   // GBK_TO_UNICODE[29568] := 16#D667;
   // GBK_TO_UNICODE[29569] := 16#8B0C;
   // GBK_TO_UNICODE[29570] := 16#D668;
   // GBK_TO_UNICODE[29571] := 16#8B0D;
   // GBK_TO_UNICODE[29572] := 16#D669;
   // GBK_TO_UNICODE[29573] := 16#8B0E;
   // GBK_TO_UNICODE[29574] := 16#D66A;
   // GBK_TO_UNICODE[29575] := 16#8B0F;
   // GBK_TO_UNICODE[29576] := 16#D66B;
   // GBK_TO_UNICODE[29577] := 16#8B10;
   // GBK_TO_UNICODE[29578] := 16#D66C;
   // GBK_TO_UNICODE[29579] := 16#8B11;
   // GBK_TO_UNICODE[29580] := 16#D66D;
   // GBK_TO_UNICODE[29581] := 16#8B12;
   // GBK_TO_UNICODE[29582] := 16#D66E;
   // GBK_TO_UNICODE[29583] := 16#8B13;
   // GBK_TO_UNICODE[29584] := 16#D66F;
   // GBK_TO_UNICODE[29585] := 16#8B14;
   // GBK_TO_UNICODE[29586] := 16#D670;
   // GBK_TO_UNICODE[29587] := 16#8B15;
   // GBK_TO_UNICODE[29588] := 16#D671;
   // GBK_TO_UNICODE[29589] := 16#8B16;
   // GBK_TO_UNICODE[29590] := 16#D672;
   // GBK_TO_UNICODE[29591] := 16#8B17;
   // GBK_TO_UNICODE[29592] := 16#D673;
   // GBK_TO_UNICODE[29593] := 16#8B18;
   // GBK_TO_UNICODE[29594] := 16#D674;
   // GBK_TO_UNICODE[29595] := 16#8B19;
   // GBK_TO_UNICODE[29596] := 16#D675;
   // GBK_TO_UNICODE[29597] := 16#8B1A;
   // GBK_TO_UNICODE[29598] := 16#D676;
   // GBK_TO_UNICODE[29599] := 16#8B1B;
   // GBK_TO_UNICODE[29600] := 16#D677;
   // GBK_TO_UNICODE[29601] := 16#8B1C;
   // GBK_TO_UNICODE[29602] := 16#D678;
   // GBK_TO_UNICODE[29603] := 16#8B1D;
   // GBK_TO_UNICODE[29604] := 16#D679;
   // GBK_TO_UNICODE[29605] := 16#8B1E;
   // GBK_TO_UNICODE[29606] := 16#D67A;
   // GBK_TO_UNICODE[29607] := 16#8B1F;
   // GBK_TO_UNICODE[29608] := 16#D67B;
   // GBK_TO_UNICODE[29609] := 16#8B20;
   // GBK_TO_UNICODE[29610] := 16#D67C;
   // GBK_TO_UNICODE[29611] := 16#8B21;
   // GBK_TO_UNICODE[29612] := 16#D67D;
   // GBK_TO_UNICODE[29613] := 16#8B22;
   // GBK_TO_UNICODE[29614] := 16#D67E;
   // GBK_TO_UNICODE[29615] := 16#8B23;
   // GBK_TO_UNICODE[29616] := 16#D680;
   // GBK_TO_UNICODE[29617] := 16#8B24;
   // GBK_TO_UNICODE[29618] := 16#D681;
   // GBK_TO_UNICODE[29619] := 16#8B25;
   // GBK_TO_UNICODE[29620] := 16#D682;
   // GBK_TO_UNICODE[29621] := 16#8B27;
   // GBK_TO_UNICODE[29622] := 16#D683;
   // GBK_TO_UNICODE[29623] := 16#8B28;
   // GBK_TO_UNICODE[29624] := 16#D684;
   // GBK_TO_UNICODE[29625] := 16#8B29;
   // GBK_TO_UNICODE[29626] := 16#D685;
   // GBK_TO_UNICODE[29627] := 16#8B2A;
   // GBK_TO_UNICODE[29628] := 16#D686;
   // GBK_TO_UNICODE[29629] := 16#8B2B;
   // GBK_TO_UNICODE[29630] := 16#D687;
   // GBK_TO_UNICODE[29631] := 16#8B2C;
   // GBK_TO_UNICODE[29632] := 16#D688;
   // GBK_TO_UNICODE[29633] := 16#8B2D;
   // GBK_TO_UNICODE[29634] := 16#D689;
   // GBK_TO_UNICODE[29635] := 16#8B2E;
   // GBK_TO_UNICODE[29636] := 16#D68A;
   // GBK_TO_UNICODE[29637] := 16#8B2F;
   // GBK_TO_UNICODE[29638] := 16#D68B;
   // GBK_TO_UNICODE[29639] := 16#8B30;
   // GBK_TO_UNICODE[29640] := 16#D68C;
   // GBK_TO_UNICODE[29641] := 16#8B31;
   // GBK_TO_UNICODE[29642] := 16#D68D;
   // GBK_TO_UNICODE[29643] := 16#8B32;
   // GBK_TO_UNICODE[29644] := 16#D68E;
   // GBK_TO_UNICODE[29645] := 16#8B33;
   // GBK_TO_UNICODE[29646] := 16#D68F;
   // GBK_TO_UNICODE[29647] := 16#8B34;
   // GBK_TO_UNICODE[29648] := 16#D690;
   // GBK_TO_UNICODE[29649] := 16#8B35;
   // GBK_TO_UNICODE[29650] := 16#D691;
   // GBK_TO_UNICODE[29651] := 16#8B36;
   // GBK_TO_UNICODE[29652] := 16#D692;
   // GBK_TO_UNICODE[29653] := 16#8B37;
   // GBK_TO_UNICODE[29654] := 16#D693;
   // GBK_TO_UNICODE[29655] := 16#8B38;
   // GBK_TO_UNICODE[29656] := 16#D694;
   // GBK_TO_UNICODE[29657] := 16#8B39;
   // GBK_TO_UNICODE[29658] := 16#D695;
   // GBK_TO_UNICODE[29659] := 16#8B3A;
   // GBK_TO_UNICODE[29660] := 16#D696;
   // GBK_TO_UNICODE[29661] := 16#8B3B;
   // GBK_TO_UNICODE[29662] := 16#D697;
   // GBK_TO_UNICODE[29663] := 16#8B3C;
   // GBK_TO_UNICODE[29664] := 16#D698;
   // GBK_TO_UNICODE[29665] := 16#8B3D;
   // GBK_TO_UNICODE[29666] := 16#D699;
   // GBK_TO_UNICODE[29667] := 16#8B3E;
   // GBK_TO_UNICODE[29668] := 16#D69A;
   // GBK_TO_UNICODE[29669] := 16#8B3F;
   // GBK_TO_UNICODE[29670] := 16#D69B;
   // GBK_TO_UNICODE[29671] := 16#8B40;
   // GBK_TO_UNICODE[29672] := 16#D69C;
   // GBK_TO_UNICODE[29673] := 16#8B41;
   // GBK_TO_UNICODE[29674] := 16#D69D;
   // GBK_TO_UNICODE[29675] := 16#8B42;
   // GBK_TO_UNICODE[29676] := 16#D69E;
   // GBK_TO_UNICODE[29677] := 16#8B43;
   // GBK_TO_UNICODE[29678] := 16#D69F;
   // GBK_TO_UNICODE[29679] := 16#8B44;
   // GBK_TO_UNICODE[29680] := 16#D6A0;
   // GBK_TO_UNICODE[29681] := 16#8B45;
   // GBK_TO_UNICODE[29682] := 16#D6A1;
   // GBK_TO_UNICODE[29683] := 16#5E27;
   // GBK_TO_UNICODE[29684] := 16#D6A2;
   // GBK_TO_UNICODE[29685] := 16#75C7;
   // GBK_TO_UNICODE[29686] := 16#D6A3;
   // GBK_TO_UNICODE[29687] := 16#90D1;
   // GBK_TO_UNICODE[29688] := 16#D6A4;
   // GBK_TO_UNICODE[29689] := 16#8BC1;
   // GBK_TO_UNICODE[29690] := 16#D6A5;
   // GBK_TO_UNICODE[29691] := 16#829D;
   // GBK_TO_UNICODE[29692] := 16#D6A6;
   // GBK_TO_UNICODE[29693] := 16#679D;
   // GBK_TO_UNICODE[29694] := 16#D6A7;
   // GBK_TO_UNICODE[29695] := 16#652F;
   // GBK_TO_UNICODE[29696] := 16#D6A8;
   // GBK_TO_UNICODE[29697] := 16#5431;
   // GBK_TO_UNICODE[29698] := 16#D6A9;
   // GBK_TO_UNICODE[29699] := 16#8718;
   // GBK_TO_UNICODE[29700] := 16#D6AA;
   // GBK_TO_UNICODE[29701] := 16#77E5;
   // GBK_TO_UNICODE[29702] := 16#D6AB;
   // GBK_TO_UNICODE[29703] := 16#80A2;
   // GBK_TO_UNICODE[29704] := 16#D6AC;
   // GBK_TO_UNICODE[29705] := 16#8102;
   // GBK_TO_UNICODE[29706] := 16#D6AD;
   // GBK_TO_UNICODE[29707] := 16#6C41;
   // GBK_TO_UNICODE[29708] := 16#D6AE;
   // GBK_TO_UNICODE[29709] := 16#4E4B;
   // GBK_TO_UNICODE[29710] := 16#D6AF;
   // GBK_TO_UNICODE[29711] := 16#7EC7;
   // GBK_TO_UNICODE[29712] := 16#D6B0;
   // GBK_TO_UNICODE[29713] := 16#804C;
   // GBK_TO_UNICODE[29714] := 16#D6B1;
   // GBK_TO_UNICODE[29715] := 16#76F4;
   // GBK_TO_UNICODE[29716] := 16#D6B2;
   // GBK_TO_UNICODE[29717] := 16#690D;
   // GBK_TO_UNICODE[29718] := 16#D6B3;
   // GBK_TO_UNICODE[29719] := 16#6B96;
   // GBK_TO_UNICODE[29720] := 16#D6B4;
   // GBK_TO_UNICODE[29721] := 16#6267;
   // GBK_TO_UNICODE[29722] := 16#D6B5;
   // GBK_TO_UNICODE[29723] := 16#503C;
   // GBK_TO_UNICODE[29724] := 16#D6B6;
   // GBK_TO_UNICODE[29725] := 16#4F84;
   // GBK_TO_UNICODE[29726] := 16#D6B7;
   // GBK_TO_UNICODE[29727] := 16#5740;
   // GBK_TO_UNICODE[29728] := 16#D6B8;
   // GBK_TO_UNICODE[29729] := 16#6307;
   // GBK_TO_UNICODE[29730] := 16#D6B9;
   // GBK_TO_UNICODE[29731] := 16#6B62;
   // GBK_TO_UNICODE[29732] := 16#D6BA;
   // GBK_TO_UNICODE[29733] := 16#8DBE;
   // GBK_TO_UNICODE[29734] := 16#D6BB;
   // GBK_TO_UNICODE[29735] := 16#53EA;
   // GBK_TO_UNICODE[29736] := 16#D6BC;
   // GBK_TO_UNICODE[29737] := 16#65E8;
   // GBK_TO_UNICODE[29738] := 16#D6BD;
   // GBK_TO_UNICODE[29739] := 16#7EB8;
   // GBK_TO_UNICODE[29740] := 16#D6BE;
   // GBK_TO_UNICODE[29741] := 16#5FD7;
   // GBK_TO_UNICODE[29742] := 16#D6BF;
   // GBK_TO_UNICODE[29743] := 16#631A;
   // GBK_TO_UNICODE[29744] := 16#D6C0;
   // GBK_TO_UNICODE[29745] := 16#63B7;
   // GBK_TO_UNICODE[29746] := 16#D6C1;
   // GBK_TO_UNICODE[29747] := 16#81F3;
   // GBK_TO_UNICODE[29748] := 16#D6C2;
   // GBK_TO_UNICODE[29749] := 16#81F4;
   // GBK_TO_UNICODE[29750] := 16#D6C3;
   // GBK_TO_UNICODE[29751] := 16#7F6E;
   // GBK_TO_UNICODE[29752] := 16#D6C4;
   // GBK_TO_UNICODE[29753] := 16#5E1C;
   // GBK_TO_UNICODE[29754] := 16#D6C5;
   // GBK_TO_UNICODE[29755] := 16#5CD9;
   // GBK_TO_UNICODE[29756] := 16#D6C6;
   // GBK_TO_UNICODE[29757] := 16#5236;
   // GBK_TO_UNICODE[29758] := 16#D6C7;
   // GBK_TO_UNICODE[29759] := 16#667A;
   // GBK_TO_UNICODE[29760] := 16#D6C8;
   // GBK_TO_UNICODE[29761] := 16#79E9;
   // GBK_TO_UNICODE[29762] := 16#D6C9;
   // GBK_TO_UNICODE[29763] := 16#7A1A;
   // GBK_TO_UNICODE[29764] := 16#D6CA;
   // GBK_TO_UNICODE[29765] := 16#8D28;
   // GBK_TO_UNICODE[29766] := 16#D6CB;
   // GBK_TO_UNICODE[29767] := 16#7099;
   // GBK_TO_UNICODE[29768] := 16#D6CC;
   // GBK_TO_UNICODE[29769] := 16#75D4;
   // GBK_TO_UNICODE[29770] := 16#D6CD;
   // GBK_TO_UNICODE[29771] := 16#6EDE;
   // GBK_TO_UNICODE[29772] := 16#D6CE;
   // GBK_TO_UNICODE[29773] := 16#6CBB;
   // GBK_TO_UNICODE[29774] := 16#D6CF;
   // GBK_TO_UNICODE[29775] := 16#7A92;
   // GBK_TO_UNICODE[29776] := 16#D6D0;
   // GBK_TO_UNICODE[29777] := 16#4E2D;
   // GBK_TO_UNICODE[29778] := 16#D6D1;
   // GBK_TO_UNICODE[29779] := 16#76C5;
   // GBK_TO_UNICODE[29780] := 16#D6D2;
   // GBK_TO_UNICODE[29781] := 16#5FE0;
   // GBK_TO_UNICODE[29782] := 16#D6D3;
   // GBK_TO_UNICODE[29783] := 16#949F;
   // GBK_TO_UNICODE[29784] := 16#D6D4;
   // GBK_TO_UNICODE[29785] := 16#8877;
   // GBK_TO_UNICODE[29786] := 16#D6D5;
   // GBK_TO_UNICODE[29787] := 16#7EC8;
   // GBK_TO_UNICODE[29788] := 16#D6D6;
   // GBK_TO_UNICODE[29789] := 16#79CD;
   // GBK_TO_UNICODE[29790] := 16#D6D7;
   // GBK_TO_UNICODE[29791] := 16#80BF;
   // GBK_TO_UNICODE[29792] := 16#D6D8;
   // GBK_TO_UNICODE[29793] := 16#91CD;
   // GBK_TO_UNICODE[29794] := 16#D6D9;
   // GBK_TO_UNICODE[29795] := 16#4EF2;
   // GBK_TO_UNICODE[29796] := 16#D6DA;
   // GBK_TO_UNICODE[29797] := 16#4F17;
   // GBK_TO_UNICODE[29798] := 16#D6DB;
   // GBK_TO_UNICODE[29799] := 16#821F;
   // GBK_TO_UNICODE[29800] := 16#D6DC;
   // GBK_TO_UNICODE[29801] := 16#5468;
   // GBK_TO_UNICODE[29802] := 16#D6DD;
   // GBK_TO_UNICODE[29803] := 16#5DDE;
   // GBK_TO_UNICODE[29804] := 16#D6DE;
   // GBK_TO_UNICODE[29805] := 16#6D32;
   // GBK_TO_UNICODE[29806] := 16#D6DF;
   // GBK_TO_UNICODE[29807] := 16#8BCC;
   // GBK_TO_UNICODE[29808] := 16#D6E0;
   // GBK_TO_UNICODE[29809] := 16#7CA5;
   // GBK_TO_UNICODE[29810] := 16#D6E1;
   // GBK_TO_UNICODE[29811] := 16#8F74;
   // GBK_TO_UNICODE[29812] := 16#D6E2;
   // GBK_TO_UNICODE[29813] := 16#8098;
   // GBK_TO_UNICODE[29814] := 16#D6E3;
   // GBK_TO_UNICODE[29815] := 16#5E1A;
   // GBK_TO_UNICODE[29816] := 16#D6E4;
   // GBK_TO_UNICODE[29817] := 16#5492;
   // GBK_TO_UNICODE[29818] := 16#D6E5;
   // GBK_TO_UNICODE[29819] := 16#76B1;
   // GBK_TO_UNICODE[29820] := 16#D6E6;
   // GBK_TO_UNICODE[29821] := 16#5B99;
   // GBK_TO_UNICODE[29822] := 16#D6E7;
   // GBK_TO_UNICODE[29823] := 16#663C;
   // GBK_TO_UNICODE[29824] := 16#D6E8;
   // GBK_TO_UNICODE[29825] := 16#9AA4;
   // GBK_TO_UNICODE[29826] := 16#D6E9;
   // GBK_TO_UNICODE[29827] := 16#73E0;
   // GBK_TO_UNICODE[29828] := 16#D6EA;
   // GBK_TO_UNICODE[29829] := 16#682A;
   // GBK_TO_UNICODE[29830] := 16#D6EB;
   // GBK_TO_UNICODE[29831] := 16#86DB;
   // GBK_TO_UNICODE[29832] := 16#D6EC;
   // GBK_TO_UNICODE[29833] := 16#6731;
   // GBK_TO_UNICODE[29834] := 16#D6ED;
   // GBK_TO_UNICODE[29835] := 16#732A;
   // GBK_TO_UNICODE[29836] := 16#D6EE;
   // GBK_TO_UNICODE[29837] := 16#8BF8;
   // GBK_TO_UNICODE[29838] := 16#D6EF;
   // GBK_TO_UNICODE[29839] := 16#8BDB;
   // GBK_TO_UNICODE[29840] := 16#D6F0;
   // GBK_TO_UNICODE[29841] := 16#9010;
   // GBK_TO_UNICODE[29842] := 16#D6F1;
   // GBK_TO_UNICODE[29843] := 16#7AF9;
   // GBK_TO_UNICODE[29844] := 16#D6F2;
   // GBK_TO_UNICODE[29845] := 16#70DB;
   // GBK_TO_UNICODE[29846] := 16#D6F3;
   // GBK_TO_UNICODE[29847] := 16#716E;
   // GBK_TO_UNICODE[29848] := 16#D6F4;
   // GBK_TO_UNICODE[29849] := 16#62C4;
   // GBK_TO_UNICODE[29850] := 16#D6F5;
   // GBK_TO_UNICODE[29851] := 16#77A9;
   // GBK_TO_UNICODE[29852] := 16#D6F6;
   // GBK_TO_UNICODE[29853] := 16#5631;
   // GBK_TO_UNICODE[29854] := 16#D6F7;
   // GBK_TO_UNICODE[29855] := 16#4E3B;
   // GBK_TO_UNICODE[29856] := 16#D6F8;
   // GBK_TO_UNICODE[29857] := 16#8457;
   // GBK_TO_UNICODE[29858] := 16#D6F9;
   // GBK_TO_UNICODE[29859] := 16#67F1;
   // GBK_TO_UNICODE[29860] := 16#D6FA;
   // GBK_TO_UNICODE[29861] := 16#52A9;
   // GBK_TO_UNICODE[29862] := 16#D6FB;
   // GBK_TO_UNICODE[29863] := 16#86C0;
   // GBK_TO_UNICODE[29864] := 16#D6FC;
   // GBK_TO_UNICODE[29865] := 16#8D2E;
   // GBK_TO_UNICODE[29866] := 16#D6FD;
   // GBK_TO_UNICODE[29867] := 16#94F8;
   // GBK_TO_UNICODE[29868] := 16#D6FE;
   // GBK_TO_UNICODE[29869] := 16#7B51;
   // GBK_TO_UNICODE[29870] := 16#D740;
   // GBK_TO_UNICODE[29871] := 16#8B46;
   // GBK_TO_UNICODE[29872] := 16#D741;
   // GBK_TO_UNICODE[29873] := 16#8B47;
   // GBK_TO_UNICODE[29874] := 16#D742;
   // GBK_TO_UNICODE[29875] := 16#8B48;
   // GBK_TO_UNICODE[29876] := 16#D743;
   // GBK_TO_UNICODE[29877] := 16#8B49;
   // GBK_TO_UNICODE[29878] := 16#D744;
   // GBK_TO_UNICODE[29879] := 16#8B4A;
   // GBK_TO_UNICODE[29880] := 16#D745;
   // GBK_TO_UNICODE[29881] := 16#8B4B;
   // GBK_TO_UNICODE[29882] := 16#D746;
   // GBK_TO_UNICODE[29883] := 16#8B4C;
   // GBK_TO_UNICODE[29884] := 16#D747;
   // GBK_TO_UNICODE[29885] := 16#8B4D;
   // GBK_TO_UNICODE[29886] := 16#D748;
   // GBK_TO_UNICODE[29887] := 16#8B4E;
   // GBK_TO_UNICODE[29888] := 16#D749;
   // GBK_TO_UNICODE[29889] := 16#8B4F;
   // GBK_TO_UNICODE[29890] := 16#D74A;
   // GBK_TO_UNICODE[29891] := 16#8B50;
   // GBK_TO_UNICODE[29892] := 16#D74B;
   // GBK_TO_UNICODE[29893] := 16#8B51;
   // GBK_TO_UNICODE[29894] := 16#D74C;
   // GBK_TO_UNICODE[29895] := 16#8B52;
   // GBK_TO_UNICODE[29896] := 16#D74D;
   // GBK_TO_UNICODE[29897] := 16#8B53;
   // GBK_TO_UNICODE[29898] := 16#D74E;
   // GBK_TO_UNICODE[29899] := 16#8B54;
   // GBK_TO_UNICODE[29900] := 16#D74F;
   // GBK_TO_UNICODE[29901] := 16#8B55;
   // GBK_TO_UNICODE[29902] := 16#D750;
   // GBK_TO_UNICODE[29903] := 16#8B56;
   // GBK_TO_UNICODE[29904] := 16#D751;
   // GBK_TO_UNICODE[29905] := 16#8B57;
   // GBK_TO_UNICODE[29906] := 16#D752;
   // GBK_TO_UNICODE[29907] := 16#8B58;
   // GBK_TO_UNICODE[29908] := 16#D753;
   // GBK_TO_UNICODE[29909] := 16#8B59;
   // GBK_TO_UNICODE[29910] := 16#D754;
   // GBK_TO_UNICODE[29911] := 16#8B5A;
   // GBK_TO_UNICODE[29912] := 16#D755;
   // GBK_TO_UNICODE[29913] := 16#8B5B;
   // GBK_TO_UNICODE[29914] := 16#D756;
   // GBK_TO_UNICODE[29915] := 16#8B5C;
   // GBK_TO_UNICODE[29916] := 16#D757;
   // GBK_TO_UNICODE[29917] := 16#8B5D;
   // GBK_TO_UNICODE[29918] := 16#D758;
   // GBK_TO_UNICODE[29919] := 16#8B5E;
   // GBK_TO_UNICODE[29920] := 16#D759;
   // GBK_TO_UNICODE[29921] := 16#8B5F;
   // GBK_TO_UNICODE[29922] := 16#D75A;
   // GBK_TO_UNICODE[29923] := 16#8B60;
   // GBK_TO_UNICODE[29924] := 16#D75B;
   // GBK_TO_UNICODE[29925] := 16#8B61;
   // GBK_TO_UNICODE[29926] := 16#D75C;
   // GBK_TO_UNICODE[29927] := 16#8B62;
   // GBK_TO_UNICODE[29928] := 16#D75D;
   // GBK_TO_UNICODE[29929] := 16#8B63;
   // GBK_TO_UNICODE[29930] := 16#D75E;
   // GBK_TO_UNICODE[29931] := 16#8B64;
   // GBK_TO_UNICODE[29932] := 16#D75F;
   // GBK_TO_UNICODE[29933] := 16#8B65;
   // GBK_TO_UNICODE[29934] := 16#D760;
   // GBK_TO_UNICODE[29935] := 16#8B67;
   // GBK_TO_UNICODE[29936] := 16#D761;
   // GBK_TO_UNICODE[29937] := 16#8B68;
   // GBK_TO_UNICODE[29938] := 16#D762;
   // GBK_TO_UNICODE[29939] := 16#8B69;
   // GBK_TO_UNICODE[29940] := 16#D763;
   // GBK_TO_UNICODE[29941] := 16#8B6A;
   // GBK_TO_UNICODE[29942] := 16#D764;
   // GBK_TO_UNICODE[29943] := 16#8B6B;
   // GBK_TO_UNICODE[29944] := 16#D765;
   // GBK_TO_UNICODE[29945] := 16#8B6D;
   // GBK_TO_UNICODE[29946] := 16#D766;
   // GBK_TO_UNICODE[29947] := 16#8B6E;
   // GBK_TO_UNICODE[29948] := 16#D767;
   // GBK_TO_UNICODE[29949] := 16#8B6F;
   // GBK_TO_UNICODE[29950] := 16#D768;
   // GBK_TO_UNICODE[29951] := 16#8B70;
   // GBK_TO_UNICODE[29952] := 16#D769;
   // GBK_TO_UNICODE[29953] := 16#8B71;
   // GBK_TO_UNICODE[29954] := 16#D76A;
   // GBK_TO_UNICODE[29955] := 16#8B72;
   // GBK_TO_UNICODE[29956] := 16#D76B;
   // GBK_TO_UNICODE[29957] := 16#8B73;
   // GBK_TO_UNICODE[29958] := 16#D76C;
   // GBK_TO_UNICODE[29959] := 16#8B74;
   // GBK_TO_UNICODE[29960] := 16#D76D;
   // GBK_TO_UNICODE[29961] := 16#8B75;
   // GBK_TO_UNICODE[29962] := 16#D76E;
   // GBK_TO_UNICODE[29963] := 16#8B76;
   // GBK_TO_UNICODE[29964] := 16#D76F;
   // GBK_TO_UNICODE[29965] := 16#8B77;
   // GBK_TO_UNICODE[29966] := 16#D770;
   // GBK_TO_UNICODE[29967] := 16#8B78;
   // GBK_TO_UNICODE[29968] := 16#D771;
   // GBK_TO_UNICODE[29969] := 16#8B79;
   // GBK_TO_UNICODE[29970] := 16#D772;
   // GBK_TO_UNICODE[29971] := 16#8B7A;
   // GBK_TO_UNICODE[29972] := 16#D773;
   // GBK_TO_UNICODE[29973] := 16#8B7B;
   // GBK_TO_UNICODE[29974] := 16#D774;
   // GBK_TO_UNICODE[29975] := 16#8B7C;
   // GBK_TO_UNICODE[29976] := 16#D775;
   // GBK_TO_UNICODE[29977] := 16#8B7D;
   // GBK_TO_UNICODE[29978] := 16#D776;
   // GBK_TO_UNICODE[29979] := 16#8B7E;
   // GBK_TO_UNICODE[29980] := 16#D777;
   // GBK_TO_UNICODE[29981] := 16#8B7F;
   // GBK_TO_UNICODE[29982] := 16#D778;
   // GBK_TO_UNICODE[29983] := 16#8B80;
   // GBK_TO_UNICODE[29984] := 16#D779;
   // GBK_TO_UNICODE[29985] := 16#8B81;
   // GBK_TO_UNICODE[29986] := 16#D77A;
   // GBK_TO_UNICODE[29987] := 16#8B82;
   // GBK_TO_UNICODE[29988] := 16#D77B;
   // GBK_TO_UNICODE[29989] := 16#8B83;
   // GBK_TO_UNICODE[29990] := 16#D77C;
   // GBK_TO_UNICODE[29991] := 16#8B84;
   // GBK_TO_UNICODE[29992] := 16#D77D;
   // GBK_TO_UNICODE[29993] := 16#8B85;
   // GBK_TO_UNICODE[29994] := 16#D77E;
   // GBK_TO_UNICODE[29995] := 16#8B86;
   // GBK_TO_UNICODE[29996] := 16#D780;
   // GBK_TO_UNICODE[29997] := 16#8B87;
   // GBK_TO_UNICODE[29998] := 16#D781;
   // GBK_TO_UNICODE[29999] := 16#8B88;
   // GBK_TO_UNICODE[30000] := 16#D782;
   // GBK_TO_UNICODE[30001] := 16#8B89;
   // GBK_TO_UNICODE[30002] := 16#D783;
   // GBK_TO_UNICODE[30003] := 16#8B8A;
   // GBK_TO_UNICODE[30004] := 16#D784;
   // GBK_TO_UNICODE[30005] := 16#8B8B;
   // GBK_TO_UNICODE[30006] := 16#D785;
   // GBK_TO_UNICODE[30007] := 16#8B8C;
   // GBK_TO_UNICODE[30008] := 16#D786;
   // GBK_TO_UNICODE[30009] := 16#8B8D;
   // GBK_TO_UNICODE[30010] := 16#D787;
   // GBK_TO_UNICODE[30011] := 16#8B8E;
   // GBK_TO_UNICODE[30012] := 16#D788;
   // GBK_TO_UNICODE[30013] := 16#8B8F;
   // GBK_TO_UNICODE[30014] := 16#D789;
   // GBK_TO_UNICODE[30015] := 16#8B90;
   // GBK_TO_UNICODE[30016] := 16#D78A;
   // GBK_TO_UNICODE[30017] := 16#8B91;
   // GBK_TO_UNICODE[30018] := 16#D78B;
   // GBK_TO_UNICODE[30019] := 16#8B92;
   // GBK_TO_UNICODE[30020] := 16#D78C;
   // GBK_TO_UNICODE[30021] := 16#8B93;
   // GBK_TO_UNICODE[30022] := 16#D78D;
   // GBK_TO_UNICODE[30023] := 16#8B94;
   // GBK_TO_UNICODE[30024] := 16#D78E;
   // GBK_TO_UNICODE[30025] := 16#8B95;
   // GBK_TO_UNICODE[30026] := 16#D78F;
   // GBK_TO_UNICODE[30027] := 16#8B96;
   // GBK_TO_UNICODE[30028] := 16#D790;
   // GBK_TO_UNICODE[30029] := 16#8B97;
   // GBK_TO_UNICODE[30030] := 16#D791;
   // GBK_TO_UNICODE[30031] := 16#8B98;
   // GBK_TO_UNICODE[30032] := 16#D792;
   // GBK_TO_UNICODE[30033] := 16#8B99;
   // GBK_TO_UNICODE[30034] := 16#D793;
   // GBK_TO_UNICODE[30035] := 16#8B9A;
   // GBK_TO_UNICODE[30036] := 16#D794;
   // GBK_TO_UNICODE[30037] := 16#8B9B;
   // GBK_TO_UNICODE[30038] := 16#D795;
   // GBK_TO_UNICODE[30039] := 16#8B9C;
   // GBK_TO_UNICODE[30040] := 16#D796;
   // GBK_TO_UNICODE[30041] := 16#8B9D;
   // GBK_TO_UNICODE[30042] := 16#D797;
   // GBK_TO_UNICODE[30043] := 16#8B9E;
   // GBK_TO_UNICODE[30044] := 16#D798;
   // GBK_TO_UNICODE[30045] := 16#8B9F;
   // GBK_TO_UNICODE[30046] := 16#D799;
   // GBK_TO_UNICODE[30047] := 16#8BAC;
   // GBK_TO_UNICODE[30048] := 16#D79A;
   // GBK_TO_UNICODE[30049] := 16#8BB1;
   // GBK_TO_UNICODE[30050] := 16#D79B;
   // GBK_TO_UNICODE[30051] := 16#8BBB;
   // GBK_TO_UNICODE[30052] := 16#D79C;
   // GBK_TO_UNICODE[30053] := 16#8BC7;
   // GBK_TO_UNICODE[30054] := 16#D79D;
   // GBK_TO_UNICODE[30055] := 16#8BD0;
   // GBK_TO_UNICODE[30056] := 16#D79E;
   // GBK_TO_UNICODE[30057] := 16#8BEA;
   // GBK_TO_UNICODE[30058] := 16#D79F;
   // GBK_TO_UNICODE[30059] := 16#8C09;
   // GBK_TO_UNICODE[30060] := 16#D7A0;
   // GBK_TO_UNICODE[30061] := 16#8C1E;
   // GBK_TO_UNICODE[30062] := 16#D7A1;
   // GBK_TO_UNICODE[30063] := 16#4F4F;
   // GBK_TO_UNICODE[30064] := 16#D7A2;
   // GBK_TO_UNICODE[30065] := 16#6CE8;
   // GBK_TO_UNICODE[30066] := 16#D7A3;
   // GBK_TO_UNICODE[30067] := 16#795D;
   // GBK_TO_UNICODE[30068] := 16#D7A4;
   // GBK_TO_UNICODE[30069] := 16#9A7B;
   // GBK_TO_UNICODE[30070] := 16#D7A5;
   // GBK_TO_UNICODE[30071] := 16#6293;
   // GBK_TO_UNICODE[30072] := 16#D7A6;
   // GBK_TO_UNICODE[30073] := 16#722A;
   // GBK_TO_UNICODE[30074] := 16#D7A7;
   // GBK_TO_UNICODE[30075] := 16#62FD;
   // GBK_TO_UNICODE[30076] := 16#D7A8;
   // GBK_TO_UNICODE[30077] := 16#4E13;
   // GBK_TO_UNICODE[30078] := 16#D7A9;
   // GBK_TO_UNICODE[30079] := 16#7816;
   // GBK_TO_UNICODE[30080] := 16#D7AA;
   // GBK_TO_UNICODE[30081] := 16#8F6C;
   // GBK_TO_UNICODE[30082] := 16#D7AB;
   // GBK_TO_UNICODE[30083] := 16#64B0;
   // GBK_TO_UNICODE[30084] := 16#D7AC;
   // GBK_TO_UNICODE[30085] := 16#8D5A;
   // GBK_TO_UNICODE[30086] := 16#D7AD;
   // GBK_TO_UNICODE[30087] := 16#7BC6;
   // GBK_TO_UNICODE[30088] := 16#D7AE;
   // GBK_TO_UNICODE[30089] := 16#6869;
   // GBK_TO_UNICODE[30090] := 16#D7AF;
   // GBK_TO_UNICODE[30091] := 16#5E84;
   // GBK_TO_UNICODE[30092] := 16#D7B0;
   // GBK_TO_UNICODE[30093] := 16#88C5;
   // GBK_TO_UNICODE[30094] := 16#D7B1;
   // GBK_TO_UNICODE[30095] := 16#5986;
   // GBK_TO_UNICODE[30096] := 16#D7B2;
   // GBK_TO_UNICODE[30097] := 16#649E;
   // GBK_TO_UNICODE[30098] := 16#D7B3;
   // GBK_TO_UNICODE[30099] := 16#58EE;
   // GBK_TO_UNICODE[30100] := 16#D7B4;
   // GBK_TO_UNICODE[30101] := 16#72B6;
   // GBK_TO_UNICODE[30102] := 16#D7B5;
   // GBK_TO_UNICODE[30103] := 16#690E;
   // GBK_TO_UNICODE[30104] := 16#D7B6;
   // GBK_TO_UNICODE[30105] := 16#9525;
   // GBK_TO_UNICODE[30106] := 16#D7B7;
   // GBK_TO_UNICODE[30107] := 16#8FFD;
   // GBK_TO_UNICODE[30108] := 16#D7B8;
   // GBK_TO_UNICODE[30109] := 16#8D58;
   // GBK_TO_UNICODE[30110] := 16#D7B9;
   // GBK_TO_UNICODE[30111] := 16#5760;
   // GBK_TO_UNICODE[30112] := 16#D7BA;
   // GBK_TO_UNICODE[30113] := 16#7F00;
   // GBK_TO_UNICODE[30114] := 16#D7BB;
   // GBK_TO_UNICODE[30115] := 16#8C06;
   // GBK_TO_UNICODE[30116] := 16#D7BC;
   // GBK_TO_UNICODE[30117] := 16#51C6;
   // GBK_TO_UNICODE[30118] := 16#D7BD;
   // GBK_TO_UNICODE[30119] := 16#6349;
   // GBK_TO_UNICODE[30120] := 16#D7BE;
   // GBK_TO_UNICODE[30121] := 16#62D9;
   // GBK_TO_UNICODE[30122] := 16#D7BF;
   // GBK_TO_UNICODE[30123] := 16#5353;
   // GBK_TO_UNICODE[30124] := 16#D7C0;
   // GBK_TO_UNICODE[30125] := 16#684C;
   // GBK_TO_UNICODE[30126] := 16#D7C1;
   // GBK_TO_UNICODE[30127] := 16#7422;
   // GBK_TO_UNICODE[30128] := 16#D7C2;
   // GBK_TO_UNICODE[30129] := 16#8301;
   // GBK_TO_UNICODE[30130] := 16#D7C3;
   // GBK_TO_UNICODE[30131] := 16#914C;
   // GBK_TO_UNICODE[30132] := 16#D7C4;
   // GBK_TO_UNICODE[30133] := 16#5544;
   // GBK_TO_UNICODE[30134] := 16#D7C5;
   // GBK_TO_UNICODE[30135] := 16#7740;
   // GBK_TO_UNICODE[30136] := 16#D7C6;
   // GBK_TO_UNICODE[30137] := 16#707C;
   // GBK_TO_UNICODE[30138] := 16#D7C7;
   // GBK_TO_UNICODE[30139] := 16#6D4A;
   // GBK_TO_UNICODE[30140] := 16#D7C8;
   // GBK_TO_UNICODE[30141] := 16#5179;
   // GBK_TO_UNICODE[30142] := 16#D7C9;
   // GBK_TO_UNICODE[30143] := 16#54A8;
   // GBK_TO_UNICODE[30144] := 16#D7CA;
   // GBK_TO_UNICODE[30145] := 16#8D44;
   // GBK_TO_UNICODE[30146] := 16#D7CB;
   // GBK_TO_UNICODE[30147] := 16#59FF;
   // GBK_TO_UNICODE[30148] := 16#D7CC;
   // GBK_TO_UNICODE[30149] := 16#6ECB;
   // GBK_TO_UNICODE[30150] := 16#D7CD;
   // GBK_TO_UNICODE[30151] := 16#6DC4;
   // GBK_TO_UNICODE[30152] := 16#D7CE;
   // GBK_TO_UNICODE[30153] := 16#5B5C;
   // GBK_TO_UNICODE[30154] := 16#D7CF;
   // GBK_TO_UNICODE[30155] := 16#7D2B;
   // GBK_TO_UNICODE[30156] := 16#D7D0;
   // GBK_TO_UNICODE[30157] := 16#4ED4;
   // GBK_TO_UNICODE[30158] := 16#D7D1;
   // GBK_TO_UNICODE[30159] := 16#7C7D;
   // GBK_TO_UNICODE[30160] := 16#D7D2;
   // GBK_TO_UNICODE[30161] := 16#6ED3;
   // GBK_TO_UNICODE[30162] := 16#D7D3;
   // GBK_TO_UNICODE[30163] := 16#5B50;
   // GBK_TO_UNICODE[30164] := 16#D7D4;
   // GBK_TO_UNICODE[30165] := 16#81EA;
   // GBK_TO_UNICODE[30166] := 16#D7D5;
   // GBK_TO_UNICODE[30167] := 16#6E0D;
   // GBK_TO_UNICODE[30168] := 16#D7D6;
   // GBK_TO_UNICODE[30169] := 16#5B57;
   // GBK_TO_UNICODE[30170] := 16#D7D7;
   // GBK_TO_UNICODE[30171] := 16#9B03;
   // GBK_TO_UNICODE[30172] := 16#D7D8;
   // GBK_TO_UNICODE[30173] := 16#68D5;
   // GBK_TO_UNICODE[30174] := 16#D7D9;
   // GBK_TO_UNICODE[30175] := 16#8E2A;
   // GBK_TO_UNICODE[30176] := 16#D7DA;
   // GBK_TO_UNICODE[30177] := 16#5B97;
   // GBK_TO_UNICODE[30178] := 16#D7DB;
   // GBK_TO_UNICODE[30179] := 16#7EFC;
   // GBK_TO_UNICODE[30180] := 16#D7DC;
   // GBK_TO_UNICODE[30181] := 16#603B;
   // GBK_TO_UNICODE[30182] := 16#D7DD;
   // GBK_TO_UNICODE[30183] := 16#7EB5;
   // GBK_TO_UNICODE[30184] := 16#D7DE;
   // GBK_TO_UNICODE[30185] := 16#90B9;
   // GBK_TO_UNICODE[30186] := 16#D7DF;
   // GBK_TO_UNICODE[30187] := 16#8D70;
   // GBK_TO_UNICODE[30188] := 16#D7E0;
   // GBK_TO_UNICODE[30189] := 16#594F;
   // GBK_TO_UNICODE[30190] := 16#D7E1;
   // GBK_TO_UNICODE[30191] := 16#63CD;
   // GBK_TO_UNICODE[30192] := 16#D7E2;
   // GBK_TO_UNICODE[30193] := 16#79DF;
   // GBK_TO_UNICODE[30194] := 16#D7E3;
   // GBK_TO_UNICODE[30195] := 16#8DB3;
   // GBK_TO_UNICODE[30196] := 16#D7E4;
   // GBK_TO_UNICODE[30197] := 16#5352;
   // GBK_TO_UNICODE[30198] := 16#D7E5;
   // GBK_TO_UNICODE[30199] := 16#65CF;
   // GBK_TO_UNICODE[30200] := 16#D7E6;
   // GBK_TO_UNICODE[30201] := 16#7956;
   // GBK_TO_UNICODE[30202] := 16#D7E7;
   // GBK_TO_UNICODE[30203] := 16#8BC5;
   // GBK_TO_UNICODE[30204] := 16#D7E8;
   // GBK_TO_UNICODE[30205] := 16#963B;
   // GBK_TO_UNICODE[30206] := 16#D7E9;
   // GBK_TO_UNICODE[30207] := 16#7EC4;
   // GBK_TO_UNICODE[30208] := 16#D7EA;
   // GBK_TO_UNICODE[30209] := 16#94BB;
   // GBK_TO_UNICODE[30210] := 16#D7EB;
   // GBK_TO_UNICODE[30211] := 16#7E82;
   // GBK_TO_UNICODE[30212] := 16#D7EC;
   // GBK_TO_UNICODE[30213] := 16#5634;
   // GBK_TO_UNICODE[30214] := 16#D7ED;
   // GBK_TO_UNICODE[30215] := 16#9189;
   // GBK_TO_UNICODE[30216] := 16#D7EE;
   // GBK_TO_UNICODE[30217] := 16#6700;
   // GBK_TO_UNICODE[30218] := 16#D7EF;
   // GBK_TO_UNICODE[30219] := 16#7F6A;
   // GBK_TO_UNICODE[30220] := 16#D7F0;
   // GBK_TO_UNICODE[30221] := 16#5C0A;
   // GBK_TO_UNICODE[30222] := 16#D7F1;
   // GBK_TO_UNICODE[30223] := 16#9075;
   // GBK_TO_UNICODE[30224] := 16#D7F2;
   // GBK_TO_UNICODE[30225] := 16#6628;
   // GBK_TO_UNICODE[30226] := 16#D7F3;
   // GBK_TO_UNICODE[30227] := 16#5DE6;
   // GBK_TO_UNICODE[30228] := 16#D7F4;
   // GBK_TO_UNICODE[30229] := 16#4F50;
   // GBK_TO_UNICODE[30230] := 16#D7F5;
   // GBK_TO_UNICODE[30231] := 16#67DE;
   // GBK_TO_UNICODE[30232] := 16#D7F6;
   // GBK_TO_UNICODE[30233] := 16#505A;
   // GBK_TO_UNICODE[30234] := 16#D7F7;
   // GBK_TO_UNICODE[30235] := 16#4F5C;
   // GBK_TO_UNICODE[30236] := 16#D7F8;
   // GBK_TO_UNICODE[30237] := 16#5750;
   // GBK_TO_UNICODE[30238] := 16#D7F9;
   // GBK_TO_UNICODE[30239] := 16#5EA7;
   // GBK_TO_UNICODE[30240] := 16#D840;
   // GBK_TO_UNICODE[30241] := 16#8C38;
   // GBK_TO_UNICODE[30242] := 16#D841;
   // GBK_TO_UNICODE[30243] := 16#8C39;
   // GBK_TO_UNICODE[30244] := 16#D842;
   // GBK_TO_UNICODE[30245] := 16#8C3A;
   // GBK_TO_UNICODE[30246] := 16#D843;
   // GBK_TO_UNICODE[30247] := 16#8C3B;
   // GBK_TO_UNICODE[30248] := 16#D844;
   // GBK_TO_UNICODE[30249] := 16#8C3C;
   // GBK_TO_UNICODE[30250] := 16#D845;
   // GBK_TO_UNICODE[30251] := 16#8C3D;
   // GBK_TO_UNICODE[30252] := 16#D846;
   // GBK_TO_UNICODE[30253] := 16#8C3E;
   // GBK_TO_UNICODE[30254] := 16#D847;
   // GBK_TO_UNICODE[30255] := 16#8C3F;
   // GBK_TO_UNICODE[30256] := 16#D848;
   // GBK_TO_UNICODE[30257] := 16#8C40;
   // GBK_TO_UNICODE[30258] := 16#D849;
   // GBK_TO_UNICODE[30259] := 16#8C42;
   // GBK_TO_UNICODE[30260] := 16#D84A;
   // GBK_TO_UNICODE[30261] := 16#8C43;
   // GBK_TO_UNICODE[30262] := 16#D84B;
   // GBK_TO_UNICODE[30263] := 16#8C44;
   // GBK_TO_UNICODE[30264] := 16#D84C;
   // GBK_TO_UNICODE[30265] := 16#8C45;
   // GBK_TO_UNICODE[30266] := 16#D84D;
   // GBK_TO_UNICODE[30267] := 16#8C48;
   // GBK_TO_UNICODE[30268] := 16#D84E;
   // GBK_TO_UNICODE[30269] := 16#8C4A;
   // GBK_TO_UNICODE[30270] := 16#D84F;
   // GBK_TO_UNICODE[30271] := 16#8C4B;
   // GBK_TO_UNICODE[30272] := 16#D850;
   // GBK_TO_UNICODE[30273] := 16#8C4D;
   // GBK_TO_UNICODE[30274] := 16#D851;
   // GBK_TO_UNICODE[30275] := 16#8C4E;
   // GBK_TO_UNICODE[30276] := 16#D852;
   // GBK_TO_UNICODE[30277] := 16#8C4F;
   // GBK_TO_UNICODE[30278] := 16#D853;
   // GBK_TO_UNICODE[30279] := 16#8C50;
   // GBK_TO_UNICODE[30280] := 16#D854;
   // GBK_TO_UNICODE[30281] := 16#8C51;
   // GBK_TO_UNICODE[30282] := 16#D855;
   // GBK_TO_UNICODE[30283] := 16#8C52;
   // GBK_TO_UNICODE[30284] := 16#D856;
   // GBK_TO_UNICODE[30285] := 16#8C53;
   // GBK_TO_UNICODE[30286] := 16#D857;
   // GBK_TO_UNICODE[30287] := 16#8C54;
   // GBK_TO_UNICODE[30288] := 16#D858;
   // GBK_TO_UNICODE[30289] := 16#8C56;
   // GBK_TO_UNICODE[30290] := 16#D859;
   // GBK_TO_UNICODE[30291] := 16#8C57;
   // GBK_TO_UNICODE[30292] := 16#D85A;
   // GBK_TO_UNICODE[30293] := 16#8C58;
   // GBK_TO_UNICODE[30294] := 16#D85B;
   // GBK_TO_UNICODE[30295] := 16#8C59;
   // GBK_TO_UNICODE[30296] := 16#D85C;
   // GBK_TO_UNICODE[30297] := 16#8C5B;
   // GBK_TO_UNICODE[30298] := 16#D85D;
   // GBK_TO_UNICODE[30299] := 16#8C5C;
   // GBK_TO_UNICODE[30300] := 16#D85E;
   // GBK_TO_UNICODE[30301] := 16#8C5D;
   // GBK_TO_UNICODE[30302] := 16#D85F;
   // GBK_TO_UNICODE[30303] := 16#8C5E;
   // GBK_TO_UNICODE[30304] := 16#D860;
   // GBK_TO_UNICODE[30305] := 16#8C5F;
   // GBK_TO_UNICODE[30306] := 16#D861;
   // GBK_TO_UNICODE[30307] := 16#8C60;
   // GBK_TO_UNICODE[30308] := 16#D862;
   // GBK_TO_UNICODE[30309] := 16#8C63;
   // GBK_TO_UNICODE[30310] := 16#D863;
   // GBK_TO_UNICODE[30311] := 16#8C64;
   // GBK_TO_UNICODE[30312] := 16#D864;
   // GBK_TO_UNICODE[30313] := 16#8C65;
   // GBK_TO_UNICODE[30314] := 16#D865;
   // GBK_TO_UNICODE[30315] := 16#8C66;
   // GBK_TO_UNICODE[30316] := 16#D866;
   // GBK_TO_UNICODE[30317] := 16#8C67;
   // GBK_TO_UNICODE[30318] := 16#D867;
   // GBK_TO_UNICODE[30319] := 16#8C68;
   // GBK_TO_UNICODE[30320] := 16#D868;
   // GBK_TO_UNICODE[30321] := 16#8C69;
   // GBK_TO_UNICODE[30322] := 16#D869;
   // GBK_TO_UNICODE[30323] := 16#8C6C;
   // GBK_TO_UNICODE[30324] := 16#D86A;
   // GBK_TO_UNICODE[30325] := 16#8C6D;
   // GBK_TO_UNICODE[30326] := 16#D86B;
   // GBK_TO_UNICODE[30327] := 16#8C6E;
   // GBK_TO_UNICODE[30328] := 16#D86C;
   // GBK_TO_UNICODE[30329] := 16#8C6F;
   // GBK_TO_UNICODE[30330] := 16#D86D;
   // GBK_TO_UNICODE[30331] := 16#8C70;
   // GBK_TO_UNICODE[30332] := 16#D86E;
   // GBK_TO_UNICODE[30333] := 16#8C71;
   // GBK_TO_UNICODE[30334] := 16#D86F;
   // GBK_TO_UNICODE[30335] := 16#8C72;
   // GBK_TO_UNICODE[30336] := 16#D870;
   // GBK_TO_UNICODE[30337] := 16#8C74;
   // GBK_TO_UNICODE[30338] := 16#D871;
   // GBK_TO_UNICODE[30339] := 16#8C75;
   // GBK_TO_UNICODE[30340] := 16#D872;
   // GBK_TO_UNICODE[30341] := 16#8C76;
   // GBK_TO_UNICODE[30342] := 16#D873;
   // GBK_TO_UNICODE[30343] := 16#8C77;
   // GBK_TO_UNICODE[30344] := 16#D874;
   // GBK_TO_UNICODE[30345] := 16#8C7B;
   // GBK_TO_UNICODE[30346] := 16#D875;
   // GBK_TO_UNICODE[30347] := 16#8C7C;
   // GBK_TO_UNICODE[30348] := 16#D876;
   // GBK_TO_UNICODE[30349] := 16#8C7D;
   // GBK_TO_UNICODE[30350] := 16#D877;
   // GBK_TO_UNICODE[30351] := 16#8C7E;
   // GBK_TO_UNICODE[30352] := 16#D878;
   // GBK_TO_UNICODE[30353] := 16#8C7F;
   // GBK_TO_UNICODE[30354] := 16#D879;
   // GBK_TO_UNICODE[30355] := 16#8C80;
   // GBK_TO_UNICODE[30356] := 16#D87A;
   // GBK_TO_UNICODE[30357] := 16#8C81;
   // GBK_TO_UNICODE[30358] := 16#D87B;
   // GBK_TO_UNICODE[30359] := 16#8C83;
   // GBK_TO_UNICODE[30360] := 16#D87C;
   // GBK_TO_UNICODE[30361] := 16#8C84;
   // GBK_TO_UNICODE[30362] := 16#D87D;
   // GBK_TO_UNICODE[30363] := 16#8C86;
   // GBK_TO_UNICODE[30364] := 16#D87E;
   // GBK_TO_UNICODE[30365] := 16#8C87;
   // GBK_TO_UNICODE[30366] := 16#D880;
   // GBK_TO_UNICODE[30367] := 16#8C88;
   // GBK_TO_UNICODE[30368] := 16#D881;
   // GBK_TO_UNICODE[30369] := 16#8C8B;
   // GBK_TO_UNICODE[30370] := 16#D882;
   // GBK_TO_UNICODE[30371] := 16#8C8D;
   // GBK_TO_UNICODE[30372] := 16#D883;
   // GBK_TO_UNICODE[30373] := 16#8C8E;
   // GBK_TO_UNICODE[30374] := 16#D884;
   // GBK_TO_UNICODE[30375] := 16#8C8F;
   // GBK_TO_UNICODE[30376] := 16#D885;
   // GBK_TO_UNICODE[30377] := 16#8C90;
   // GBK_TO_UNICODE[30378] := 16#D886;
   // GBK_TO_UNICODE[30379] := 16#8C91;
   // GBK_TO_UNICODE[30380] := 16#D887;
   // GBK_TO_UNICODE[30381] := 16#8C92;
   // GBK_TO_UNICODE[30382] := 16#D888;
   // GBK_TO_UNICODE[30383] := 16#8C93;
   // GBK_TO_UNICODE[30384] := 16#D889;
   // GBK_TO_UNICODE[30385] := 16#8C95;
   // GBK_TO_UNICODE[30386] := 16#D88A;
   // GBK_TO_UNICODE[30387] := 16#8C96;
   // GBK_TO_UNICODE[30388] := 16#D88B;
   // GBK_TO_UNICODE[30389] := 16#8C97;
   // GBK_TO_UNICODE[30390] := 16#D88C;
   // GBK_TO_UNICODE[30391] := 16#8C99;
   // GBK_TO_UNICODE[30392] := 16#D88D;
   // GBK_TO_UNICODE[30393] := 16#8C9A;
   // GBK_TO_UNICODE[30394] := 16#D88E;
   // GBK_TO_UNICODE[30395] := 16#8C9B;
   // GBK_TO_UNICODE[30396] := 16#D88F;
   // GBK_TO_UNICODE[30397] := 16#8C9C;
   // GBK_TO_UNICODE[30398] := 16#D890;
   // GBK_TO_UNICODE[30399] := 16#8C9D;
   // GBK_TO_UNICODE[30400] := 16#D891;
   // GBK_TO_UNICODE[30401] := 16#8C9E;
   // GBK_TO_UNICODE[30402] := 16#D892;
   // GBK_TO_UNICODE[30403] := 16#8C9F;
   // GBK_TO_UNICODE[30404] := 16#D893;
   // GBK_TO_UNICODE[30405] := 16#8CA0;
   // GBK_TO_UNICODE[30406] := 16#D894;
   // GBK_TO_UNICODE[30407] := 16#8CA1;
   // GBK_TO_UNICODE[30408] := 16#D895;
   // GBK_TO_UNICODE[30409] := 16#8CA2;
   // GBK_TO_UNICODE[30410] := 16#D896;
   // GBK_TO_UNICODE[30411] := 16#8CA3;
   // GBK_TO_UNICODE[30412] := 16#D897;
   // GBK_TO_UNICODE[30413] := 16#8CA4;
   // GBK_TO_UNICODE[30414] := 16#D898;
   // GBK_TO_UNICODE[30415] := 16#8CA5;
   // GBK_TO_UNICODE[30416] := 16#D899;
   // GBK_TO_UNICODE[30417] := 16#8CA6;
   // GBK_TO_UNICODE[30418] := 16#D89A;
   // GBK_TO_UNICODE[30419] := 16#8CA7;
   // GBK_TO_UNICODE[30420] := 16#D89B;
   // GBK_TO_UNICODE[30421] := 16#8CA8;
   // GBK_TO_UNICODE[30422] := 16#D89C;
   // GBK_TO_UNICODE[30423] := 16#8CA9;
   // GBK_TO_UNICODE[30424] := 16#D89D;
   // GBK_TO_UNICODE[30425] := 16#8CAA;
   // GBK_TO_UNICODE[30426] := 16#D89E;
   // GBK_TO_UNICODE[30427] := 16#8CAB;
   // GBK_TO_UNICODE[30428] := 16#D89F;
   // GBK_TO_UNICODE[30429] := 16#8CAC;
   // GBK_TO_UNICODE[30430] := 16#D8A0;
   // GBK_TO_UNICODE[30431] := 16#8CAD;
   // GBK_TO_UNICODE[30432] := 16#D8A1;
   // GBK_TO_UNICODE[30433] := 16#4E8D;
   // GBK_TO_UNICODE[30434] := 16#D8A2;
   // GBK_TO_UNICODE[30435] := 16#4E0C;
   // GBK_TO_UNICODE[30436] := 16#D8A3;
   // GBK_TO_UNICODE[30437] := 16#5140;
   // GBK_TO_UNICODE[30438] := 16#D8A4;
   // GBK_TO_UNICODE[30439] := 16#4E10;
   // GBK_TO_UNICODE[30440] := 16#D8A5;
   // GBK_TO_UNICODE[30441] := 16#5EFF;
   // GBK_TO_UNICODE[30442] := 16#D8A6;
   // GBK_TO_UNICODE[30443] := 16#5345;
   // GBK_TO_UNICODE[30444] := 16#D8A7;
   // GBK_TO_UNICODE[30445] := 16#4E15;
   // GBK_TO_UNICODE[30446] := 16#D8A8;
   // GBK_TO_UNICODE[30447] := 16#4E98;
   // GBK_TO_UNICODE[30448] := 16#D8A9;
   // GBK_TO_UNICODE[30449] := 16#4E1E;
   // GBK_TO_UNICODE[30450] := 16#D8AA;
   // GBK_TO_UNICODE[30451] := 16#9B32;
   // GBK_TO_UNICODE[30452] := 16#D8AB;
   // GBK_TO_UNICODE[30453] := 16#5B6C;
   // GBK_TO_UNICODE[30454] := 16#D8AC;
   // GBK_TO_UNICODE[30455] := 16#5669;
   // GBK_TO_UNICODE[30456] := 16#D8AD;
   // GBK_TO_UNICODE[30457] := 16#4E28;
   // GBK_TO_UNICODE[30458] := 16#D8AE;
   // GBK_TO_UNICODE[30459] := 16#79BA;
   // GBK_TO_UNICODE[30460] := 16#D8AF;
   // GBK_TO_UNICODE[30461] := 16#4E3F;
   // GBK_TO_UNICODE[30462] := 16#D8B0;
   // GBK_TO_UNICODE[30463] := 16#5315;
   // GBK_TO_UNICODE[30464] := 16#D8B1;
   // GBK_TO_UNICODE[30465] := 16#4E47;
   // GBK_TO_UNICODE[30466] := 16#D8B2;
   // GBK_TO_UNICODE[30467] := 16#592D;
   // GBK_TO_UNICODE[30468] := 16#D8B3;
   // GBK_TO_UNICODE[30469] := 16#723B;
   // GBK_TO_UNICODE[30470] := 16#D8B4;
   // GBK_TO_UNICODE[30471] := 16#536E;
   // GBK_TO_UNICODE[30472] := 16#D8B5;
   // GBK_TO_UNICODE[30473] := 16#6C10;
   // GBK_TO_UNICODE[30474] := 16#D8B6;
   // GBK_TO_UNICODE[30475] := 16#56DF;
   // GBK_TO_UNICODE[30476] := 16#D8B7;
   // GBK_TO_UNICODE[30477] := 16#80E4;
   // GBK_TO_UNICODE[30478] := 16#D8B8;
   // GBK_TO_UNICODE[30479] := 16#9997;
   // GBK_TO_UNICODE[30480] := 16#D8B9;
   // GBK_TO_UNICODE[30481] := 16#6BD3;
   // GBK_TO_UNICODE[30482] := 16#D8BA;
   // GBK_TO_UNICODE[30483] := 16#777E;
   // GBK_TO_UNICODE[30484] := 16#D8BB;
   // GBK_TO_UNICODE[30485] := 16#9F17;
   // GBK_TO_UNICODE[30486] := 16#D8BC;
   // GBK_TO_UNICODE[30487] := 16#4E36;
   // GBK_TO_UNICODE[30488] := 16#D8BD;
   // GBK_TO_UNICODE[30489] := 16#4E9F;
   // GBK_TO_UNICODE[30490] := 16#D8BE;
   // GBK_TO_UNICODE[30491] := 16#9F10;
   // GBK_TO_UNICODE[30492] := 16#D8BF;
   // GBK_TO_UNICODE[30493] := 16#4E5C;
   // GBK_TO_UNICODE[30494] := 16#D8C0;
   // GBK_TO_UNICODE[30495] := 16#4E69;
   // GBK_TO_UNICODE[30496] := 16#D8C1;
   // GBK_TO_UNICODE[30497] := 16#4E93;
   // GBK_TO_UNICODE[30498] := 16#D8C2;
   // GBK_TO_UNICODE[30499] := 16#8288;
   // GBK_TO_UNICODE[30500] := 16#D8C3;
   // GBK_TO_UNICODE[30501] := 16#5B5B;
   // GBK_TO_UNICODE[30502] := 16#D8C4;
   // GBK_TO_UNICODE[30503] := 16#556C;
   // GBK_TO_UNICODE[30504] := 16#D8C5;
   // GBK_TO_UNICODE[30505] := 16#560F;
   // GBK_TO_UNICODE[30506] := 16#D8C6;
   // GBK_TO_UNICODE[30507] := 16#4EC4;
   // GBK_TO_UNICODE[30508] := 16#D8C7;
   // GBK_TO_UNICODE[30509] := 16#538D;
   // GBK_TO_UNICODE[30510] := 16#D8C8;
   // GBK_TO_UNICODE[30511] := 16#539D;
   // GBK_TO_UNICODE[30512] := 16#D8C9;
   // GBK_TO_UNICODE[30513] := 16#53A3;
   // GBK_TO_UNICODE[30514] := 16#D8CA;
   // GBK_TO_UNICODE[30515] := 16#53A5;
   // GBK_TO_UNICODE[30516] := 16#D8CB;
   // GBK_TO_UNICODE[30517] := 16#53AE;
   // GBK_TO_UNICODE[30518] := 16#D8CC;
   // GBK_TO_UNICODE[30519] := 16#9765;
   // GBK_TO_UNICODE[30520] := 16#D8CD;
   // GBK_TO_UNICODE[30521] := 16#8D5D;
   // GBK_TO_UNICODE[30522] := 16#D8CE;
   // GBK_TO_UNICODE[30523] := 16#531A;
   // GBK_TO_UNICODE[30524] := 16#D8CF;
   // GBK_TO_UNICODE[30525] := 16#53F5;
   // GBK_TO_UNICODE[30526] := 16#D8D0;
   // GBK_TO_UNICODE[30527] := 16#5326;
   // GBK_TO_UNICODE[30528] := 16#D8D1;
   // GBK_TO_UNICODE[30529] := 16#532E;
   // GBK_TO_UNICODE[30530] := 16#D8D2;
   // GBK_TO_UNICODE[30531] := 16#533E;
   // GBK_TO_UNICODE[30532] := 16#D8D3;
   // GBK_TO_UNICODE[30533] := 16#8D5C;
   // GBK_TO_UNICODE[30534] := 16#D8D4;
   // GBK_TO_UNICODE[30535] := 16#5366;
   // GBK_TO_UNICODE[30536] := 16#D8D5;
   // GBK_TO_UNICODE[30537] := 16#5363;
   // GBK_TO_UNICODE[30538] := 16#D8D6;
   // GBK_TO_UNICODE[30539] := 16#5202;
   // GBK_TO_UNICODE[30540] := 16#D8D7;
   // GBK_TO_UNICODE[30541] := 16#5208;
   // GBK_TO_UNICODE[30542] := 16#D8D8;
   // GBK_TO_UNICODE[30543] := 16#520E;
   // GBK_TO_UNICODE[30544] := 16#D8D9;
   // GBK_TO_UNICODE[30545] := 16#522D;
   // GBK_TO_UNICODE[30546] := 16#D8DA;
   // GBK_TO_UNICODE[30547] := 16#5233;
   // GBK_TO_UNICODE[30548] := 16#D8DB;
   // GBK_TO_UNICODE[30549] := 16#523F;
   // GBK_TO_UNICODE[30550] := 16#D8DC;
   // GBK_TO_UNICODE[30551] := 16#5240;
   // GBK_TO_UNICODE[30552] := 16#D8DD;
   // GBK_TO_UNICODE[30553] := 16#524C;
   // GBK_TO_UNICODE[30554] := 16#D8DE;
   // GBK_TO_UNICODE[30555] := 16#525E;
   // GBK_TO_UNICODE[30556] := 16#D8DF;
   // GBK_TO_UNICODE[30557] := 16#5261;
   // GBK_TO_UNICODE[30558] := 16#D8E0;
   // GBK_TO_UNICODE[30559] := 16#525C;
   // GBK_TO_UNICODE[30560] := 16#D8E1;
   // GBK_TO_UNICODE[30561] := 16#84AF;
   // GBK_TO_UNICODE[30562] := 16#D8E2;
   // GBK_TO_UNICODE[30563] := 16#527D;
   // GBK_TO_UNICODE[30564] := 16#D8E3;
   // GBK_TO_UNICODE[30565] := 16#5282;
   // GBK_TO_UNICODE[30566] := 16#D8E4;
   // GBK_TO_UNICODE[30567] := 16#5281;
   // GBK_TO_UNICODE[30568] := 16#D8E5;
   // GBK_TO_UNICODE[30569] := 16#5290;
   // GBK_TO_UNICODE[30570] := 16#D8E6;
   // GBK_TO_UNICODE[30571] := 16#5293;
   // GBK_TO_UNICODE[30572] := 16#D8E7;
   // GBK_TO_UNICODE[30573] := 16#5182;
   // GBK_TO_UNICODE[30574] := 16#D8E8;
   // GBK_TO_UNICODE[30575] := 16#7F54;
   // GBK_TO_UNICODE[30576] := 16#D8E9;
   // GBK_TO_UNICODE[30577] := 16#4EBB;
   // GBK_TO_UNICODE[30578] := 16#D8EA;
   // GBK_TO_UNICODE[30579] := 16#4EC3;
   // GBK_TO_UNICODE[30580] := 16#D8EB;
   // GBK_TO_UNICODE[30581] := 16#4EC9;
   // GBK_TO_UNICODE[30582] := 16#D8EC;
   // GBK_TO_UNICODE[30583] := 16#4EC2;
   // GBK_TO_UNICODE[30584] := 16#D8ED;
   // GBK_TO_UNICODE[30585] := 16#4EE8;
   // GBK_TO_UNICODE[30586] := 16#D8EE;
   // GBK_TO_UNICODE[30587] := 16#4EE1;
   // GBK_TO_UNICODE[30588] := 16#D8EF;
   // GBK_TO_UNICODE[30589] := 16#4EEB;
   // GBK_TO_UNICODE[30590] := 16#D8F0;
   // GBK_TO_UNICODE[30591] := 16#4EDE;
   // GBK_TO_UNICODE[30592] := 16#D8F1;
   // GBK_TO_UNICODE[30593] := 16#4F1B;
   // GBK_TO_UNICODE[30594] := 16#D8F2;
   // GBK_TO_UNICODE[30595] := 16#4EF3;
   // GBK_TO_UNICODE[30596] := 16#D8F3;
   // GBK_TO_UNICODE[30597] := 16#4F22;
   // GBK_TO_UNICODE[30598] := 16#D8F4;
   // GBK_TO_UNICODE[30599] := 16#4F64;
   // GBK_TO_UNICODE[30600] := 16#D8F5;
   // GBK_TO_UNICODE[30601] := 16#4EF5;
   // GBK_TO_UNICODE[30602] := 16#D8F6;
   // GBK_TO_UNICODE[30603] := 16#4F25;
   // GBK_TO_UNICODE[30604] := 16#D8F7;
   // GBK_TO_UNICODE[30605] := 16#4F27;
   // GBK_TO_UNICODE[30606] := 16#D8F8;
   // GBK_TO_UNICODE[30607] := 16#4F09;
   // GBK_TO_UNICODE[30608] := 16#D8F9;
   // GBK_TO_UNICODE[30609] := 16#4F2B;
   // GBK_TO_UNICODE[30610] := 16#D8FA;
   // GBK_TO_UNICODE[30611] := 16#4F5E;
   // GBK_TO_UNICODE[30612] := 16#D8FB;
   // GBK_TO_UNICODE[30613] := 16#4F67;
   // GBK_TO_UNICODE[30614] := 16#D8FC;
   // GBK_TO_UNICODE[30615] := 16#6538;
   // GBK_TO_UNICODE[30616] := 16#D8FD;
   // GBK_TO_UNICODE[30617] := 16#4F5A;
   // GBK_TO_UNICODE[30618] := 16#D8FE;
   // GBK_TO_UNICODE[30619] := 16#4F5D;
   // GBK_TO_UNICODE[30620] := 16#D940;
   // GBK_TO_UNICODE[30621] := 16#8CAE;
   // GBK_TO_UNICODE[30622] := 16#D941;
   // GBK_TO_UNICODE[30623] := 16#8CAF;
   // GBK_TO_UNICODE[30624] := 16#D942;
   // GBK_TO_UNICODE[30625] := 16#8CB0;
   // GBK_TO_UNICODE[30626] := 16#D943;
   // GBK_TO_UNICODE[30627] := 16#8CB1;
   // GBK_TO_UNICODE[30628] := 16#D944;
   // GBK_TO_UNICODE[30629] := 16#8CB2;
   // GBK_TO_UNICODE[30630] := 16#D945;
   // GBK_TO_UNICODE[30631] := 16#8CB3;
   // GBK_TO_UNICODE[30632] := 16#D946;
   // GBK_TO_UNICODE[30633] := 16#8CB4;
   // GBK_TO_UNICODE[30634] := 16#D947;
   // GBK_TO_UNICODE[30635] := 16#8CB5;
   // GBK_TO_UNICODE[30636] := 16#D948;
   // GBK_TO_UNICODE[30637] := 16#8CB6;
   // GBK_TO_UNICODE[30638] := 16#D949;
   // GBK_TO_UNICODE[30639] := 16#8CB7;
   // GBK_TO_UNICODE[30640] := 16#D94A;
   // GBK_TO_UNICODE[30641] := 16#8CB8;
   // GBK_TO_UNICODE[30642] := 16#D94B;
   // GBK_TO_UNICODE[30643] := 16#8CB9;
   // GBK_TO_UNICODE[30644] := 16#D94C;
   // GBK_TO_UNICODE[30645] := 16#8CBA;
   // GBK_TO_UNICODE[30646] := 16#D94D;
   // GBK_TO_UNICODE[30647] := 16#8CBB;
   // GBK_TO_UNICODE[30648] := 16#D94E;
   // GBK_TO_UNICODE[30649] := 16#8CBC;
   // GBK_TO_UNICODE[30650] := 16#D94F;
   // GBK_TO_UNICODE[30651] := 16#8CBD;
   // GBK_TO_UNICODE[30652] := 16#D950;
   // GBK_TO_UNICODE[30653] := 16#8CBE;
   // GBK_TO_UNICODE[30654] := 16#D951;
   // GBK_TO_UNICODE[30655] := 16#8CBF;
   // GBK_TO_UNICODE[30656] := 16#D952;
   // GBK_TO_UNICODE[30657] := 16#8CC0;
   // GBK_TO_UNICODE[30658] := 16#D953;
   // GBK_TO_UNICODE[30659] := 16#8CC1;
   // GBK_TO_UNICODE[30660] := 16#D954;
   // GBK_TO_UNICODE[30661] := 16#8CC2;
   // GBK_TO_UNICODE[30662] := 16#D955;
   // GBK_TO_UNICODE[30663] := 16#8CC3;
   // GBK_TO_UNICODE[30664] := 16#D956;
   // GBK_TO_UNICODE[30665] := 16#8CC4;
   // GBK_TO_UNICODE[30666] := 16#D957;
   // GBK_TO_UNICODE[30667] := 16#8CC5;
   // GBK_TO_UNICODE[30668] := 16#D958;
   // GBK_TO_UNICODE[30669] := 16#8CC6;
   // GBK_TO_UNICODE[30670] := 16#D959;
   // GBK_TO_UNICODE[30671] := 16#8CC7;
   // GBK_TO_UNICODE[30672] := 16#D95A;
   // GBK_TO_UNICODE[30673] := 16#8CC8;
   // GBK_TO_UNICODE[30674] := 16#D95B;
   // GBK_TO_UNICODE[30675] := 16#8CC9;
   // GBK_TO_UNICODE[30676] := 16#D95C;
   // GBK_TO_UNICODE[30677] := 16#8CCA;
   // GBK_TO_UNICODE[30678] := 16#D95D;
   // GBK_TO_UNICODE[30679] := 16#8CCB;
   // GBK_TO_UNICODE[30680] := 16#D95E;
   // GBK_TO_UNICODE[30681] := 16#8CCC;
   // GBK_TO_UNICODE[30682] := 16#D95F;
   // GBK_TO_UNICODE[30683] := 16#8CCD;
   // GBK_TO_UNICODE[30684] := 16#D960;
   // GBK_TO_UNICODE[30685] := 16#8CCE;
   // GBK_TO_UNICODE[30686] := 16#D961;
   // GBK_TO_UNICODE[30687] := 16#8CCF;
   // GBK_TO_UNICODE[30688] := 16#D962;
   // GBK_TO_UNICODE[30689] := 16#8CD0;
   // GBK_TO_UNICODE[30690] := 16#D963;
   // GBK_TO_UNICODE[30691] := 16#8CD1;
   // GBK_TO_UNICODE[30692] := 16#D964;
   // GBK_TO_UNICODE[30693] := 16#8CD2;
   // GBK_TO_UNICODE[30694] := 16#D965;
   // GBK_TO_UNICODE[30695] := 16#8CD3;
   // GBK_TO_UNICODE[30696] := 16#D966;
   // GBK_TO_UNICODE[30697] := 16#8CD4;
   // GBK_TO_UNICODE[30698] := 16#D967;
   // GBK_TO_UNICODE[30699] := 16#8CD5;
   // GBK_TO_UNICODE[30700] := 16#D968;
   // GBK_TO_UNICODE[30701] := 16#8CD6;
   // GBK_TO_UNICODE[30702] := 16#D969;
   // GBK_TO_UNICODE[30703] := 16#8CD7;
   // GBK_TO_UNICODE[30704] := 16#D96A;
   // GBK_TO_UNICODE[30705] := 16#8CD8;
   // GBK_TO_UNICODE[30706] := 16#D96B;
   // GBK_TO_UNICODE[30707] := 16#8CD9;
   // GBK_TO_UNICODE[30708] := 16#D96C;
   // GBK_TO_UNICODE[30709] := 16#8CDA;
   // GBK_TO_UNICODE[30710] := 16#D96D;
   // GBK_TO_UNICODE[30711] := 16#8CDB;
   // GBK_TO_UNICODE[30712] := 16#D96E;
   // GBK_TO_UNICODE[30713] := 16#8CDC;
   // GBK_TO_UNICODE[30714] := 16#D96F;
   // GBK_TO_UNICODE[30715] := 16#8CDD;
   // GBK_TO_UNICODE[30716] := 16#D970;
   // GBK_TO_UNICODE[30717] := 16#8CDE;
   // GBK_TO_UNICODE[30718] := 16#D971;
   // GBK_TO_UNICODE[30719] := 16#8CDF;
   // GBK_TO_UNICODE[30720] := 16#D972;
   // GBK_TO_UNICODE[30721] := 16#8CE0;
   // GBK_TO_UNICODE[30722] := 16#D973;
   // GBK_TO_UNICODE[30723] := 16#8CE1;
   // GBK_TO_UNICODE[30724] := 16#D974;
   // GBK_TO_UNICODE[30725] := 16#8CE2;
   // GBK_TO_UNICODE[30726] := 16#D975;
   // GBK_TO_UNICODE[30727] := 16#8CE3;
   // GBK_TO_UNICODE[30728] := 16#D976;
   // GBK_TO_UNICODE[30729] := 16#8CE4;
   // GBK_TO_UNICODE[30730] := 16#D977;
   // GBK_TO_UNICODE[30731] := 16#8CE5;
   // GBK_TO_UNICODE[30732] := 16#D978;
   // GBK_TO_UNICODE[30733] := 16#8CE6;
   // GBK_TO_UNICODE[30734] := 16#D979;
   // GBK_TO_UNICODE[30735] := 16#8CE7;
   // GBK_TO_UNICODE[30736] := 16#D97A;
   // GBK_TO_UNICODE[30737] := 16#8CE8;
   // GBK_TO_UNICODE[30738] := 16#D97B;
   // GBK_TO_UNICODE[30739] := 16#8CE9;
   // GBK_TO_UNICODE[30740] := 16#D97C;
   // GBK_TO_UNICODE[30741] := 16#8CEA;
   // GBK_TO_UNICODE[30742] := 16#D97D;
   // GBK_TO_UNICODE[30743] := 16#8CEB;
   // GBK_TO_UNICODE[30744] := 16#D97E;
   // GBK_TO_UNICODE[30745] := 16#8CEC;
   // GBK_TO_UNICODE[30746] := 16#D980;
   // GBK_TO_UNICODE[30747] := 16#8CED;
   // GBK_TO_UNICODE[30748] := 16#D981;
   // GBK_TO_UNICODE[30749] := 16#8CEE;
   // GBK_TO_UNICODE[30750] := 16#D982;
   // GBK_TO_UNICODE[30751] := 16#8CEF;
   // GBK_TO_UNICODE[30752] := 16#D983;
   // GBK_TO_UNICODE[30753] := 16#8CF0;
   // GBK_TO_UNICODE[30754] := 16#D984;
   // GBK_TO_UNICODE[30755] := 16#8CF1;
   // GBK_TO_UNICODE[30756] := 16#D985;
   // GBK_TO_UNICODE[30757] := 16#8CF2;
   // GBK_TO_UNICODE[30758] := 16#D986;
   // GBK_TO_UNICODE[30759] := 16#8CF3;
   // GBK_TO_UNICODE[30760] := 16#D987;
   // GBK_TO_UNICODE[30761] := 16#8CF4;
   // GBK_TO_UNICODE[30762] := 16#D988;
   // GBK_TO_UNICODE[30763] := 16#8CF5;
   // GBK_TO_UNICODE[30764] := 16#D989;
   // GBK_TO_UNICODE[30765] := 16#8CF6;
   // GBK_TO_UNICODE[30766] := 16#D98A;
   // GBK_TO_UNICODE[30767] := 16#8CF7;
   // GBK_TO_UNICODE[30768] := 16#D98B;
   // GBK_TO_UNICODE[30769] := 16#8CF8;
   // GBK_TO_UNICODE[30770] := 16#D98C;
   // GBK_TO_UNICODE[30771] := 16#8CF9;
   // GBK_TO_UNICODE[30772] := 16#D98D;
   // GBK_TO_UNICODE[30773] := 16#8CFA;
   // GBK_TO_UNICODE[30774] := 16#D98E;
   // GBK_TO_UNICODE[30775] := 16#8CFB;
   // GBK_TO_UNICODE[30776] := 16#D98F;
   // GBK_TO_UNICODE[30777] := 16#8CFC;
   // GBK_TO_UNICODE[30778] := 16#D990;
   // GBK_TO_UNICODE[30779] := 16#8CFD;
   // GBK_TO_UNICODE[30780] := 16#D991;
   // GBK_TO_UNICODE[30781] := 16#8CFE;
   // GBK_TO_UNICODE[30782] := 16#D992;
   // GBK_TO_UNICODE[30783] := 16#8CFF;
   // GBK_TO_UNICODE[30784] := 16#D993;
   // GBK_TO_UNICODE[30785] := 16#8D00;
   // GBK_TO_UNICODE[30786] := 16#D994;
   // GBK_TO_UNICODE[30787] := 16#8D01;
   // GBK_TO_UNICODE[30788] := 16#D995;
   // GBK_TO_UNICODE[30789] := 16#8D02;
   // GBK_TO_UNICODE[30790] := 16#D996;
   // GBK_TO_UNICODE[30791] := 16#8D03;
   // GBK_TO_UNICODE[30792] := 16#D997;
   // GBK_TO_UNICODE[30793] := 16#8D04;
   // GBK_TO_UNICODE[30794] := 16#D998;
   // GBK_TO_UNICODE[30795] := 16#8D05;
   // GBK_TO_UNICODE[30796] := 16#D999;
   // GBK_TO_UNICODE[30797] := 16#8D06;
   // GBK_TO_UNICODE[30798] := 16#D99A;
   // GBK_TO_UNICODE[30799] := 16#8D07;
   // GBK_TO_UNICODE[30800] := 16#D99B;
   // GBK_TO_UNICODE[30801] := 16#8D08;
   // GBK_TO_UNICODE[30802] := 16#D99C;
   // GBK_TO_UNICODE[30803] := 16#8D09;
   // GBK_TO_UNICODE[30804] := 16#D99D;
   // GBK_TO_UNICODE[30805] := 16#8D0A;
   // GBK_TO_UNICODE[30806] := 16#D99E;
   // GBK_TO_UNICODE[30807] := 16#8D0B;
   // GBK_TO_UNICODE[30808] := 16#D99F;
   // GBK_TO_UNICODE[30809] := 16#8D0C;
   // GBK_TO_UNICODE[30810] := 16#D9A0;
   // GBK_TO_UNICODE[30811] := 16#8D0D;
   // GBK_TO_UNICODE[30812] := 16#D9A1;
   // GBK_TO_UNICODE[30813] := 16#4F5F;
   // GBK_TO_UNICODE[30814] := 16#D9A2;
   // GBK_TO_UNICODE[30815] := 16#4F57;
   // GBK_TO_UNICODE[30816] := 16#D9A3;
   // GBK_TO_UNICODE[30817] := 16#4F32;
   // GBK_TO_UNICODE[30818] := 16#D9A4;
   // GBK_TO_UNICODE[30819] := 16#4F3D;
   // GBK_TO_UNICODE[30820] := 16#D9A5;
   // GBK_TO_UNICODE[30821] := 16#4F76;
   // GBK_TO_UNICODE[30822] := 16#D9A6;
   // GBK_TO_UNICODE[30823] := 16#4F74;
   // GBK_TO_UNICODE[30824] := 16#D9A7;
   // GBK_TO_UNICODE[30825] := 16#4F91;
   // GBK_TO_UNICODE[30826] := 16#D9A8;
   // GBK_TO_UNICODE[30827] := 16#4F89;
   // GBK_TO_UNICODE[30828] := 16#D9A9;
   // GBK_TO_UNICODE[30829] := 16#4F83;
   // GBK_TO_UNICODE[30830] := 16#D9AA;
   // GBK_TO_UNICODE[30831] := 16#4F8F;
   // GBK_TO_UNICODE[30832] := 16#D9AB;
   // GBK_TO_UNICODE[30833] := 16#4F7E;
   // GBK_TO_UNICODE[30834] := 16#D9AC;
   // GBK_TO_UNICODE[30835] := 16#4F7B;
   // GBK_TO_UNICODE[30836] := 16#D9AD;
   // GBK_TO_UNICODE[30837] := 16#4FAA;
   // GBK_TO_UNICODE[30838] := 16#D9AE;
   // GBK_TO_UNICODE[30839] := 16#4F7C;
   // GBK_TO_UNICODE[30840] := 16#D9AF;
   // GBK_TO_UNICODE[30841] := 16#4FAC;
   // GBK_TO_UNICODE[30842] := 16#D9B0;
   // GBK_TO_UNICODE[30843] := 16#4F94;
   // GBK_TO_UNICODE[30844] := 16#D9B1;
   // GBK_TO_UNICODE[30845] := 16#4FE6;
   // GBK_TO_UNICODE[30846] := 16#D9B2;
   // GBK_TO_UNICODE[30847] := 16#4FE8;
   // GBK_TO_UNICODE[30848] := 16#D9B3;
   // GBK_TO_UNICODE[30849] := 16#4FEA;
   // GBK_TO_UNICODE[30850] := 16#D9B4;
   // GBK_TO_UNICODE[30851] := 16#4FC5;
   // GBK_TO_UNICODE[30852] := 16#D9B5;
   // GBK_TO_UNICODE[30853] := 16#4FDA;
   // GBK_TO_UNICODE[30854] := 16#D9B6;
   // GBK_TO_UNICODE[30855] := 16#4FE3;
   // GBK_TO_UNICODE[30856] := 16#D9B7;
   // GBK_TO_UNICODE[30857] := 16#4FDC;
   // GBK_TO_UNICODE[30858] := 16#D9B8;
   // GBK_TO_UNICODE[30859] := 16#4FD1;
   // GBK_TO_UNICODE[30860] := 16#D9B9;
   // GBK_TO_UNICODE[30861] := 16#4FDF;
   // GBK_TO_UNICODE[30862] := 16#D9BA;
   // GBK_TO_UNICODE[30863] := 16#4FF8;
   // GBK_TO_UNICODE[30864] := 16#D9BB;
   // GBK_TO_UNICODE[30865] := 16#5029;
   // GBK_TO_UNICODE[30866] := 16#D9BC;
   // GBK_TO_UNICODE[30867] := 16#504C;
   // GBK_TO_UNICODE[30868] := 16#D9BD;
   // GBK_TO_UNICODE[30869] := 16#4FF3;
   // GBK_TO_UNICODE[30870] := 16#D9BE;
   // GBK_TO_UNICODE[30871] := 16#502C;
   // GBK_TO_UNICODE[30872] := 16#D9BF;
   // GBK_TO_UNICODE[30873] := 16#500F;
   // GBK_TO_UNICODE[30874] := 16#D9C0;
   // GBK_TO_UNICODE[30875] := 16#502E;
   // GBK_TO_UNICODE[30876] := 16#D9C1;
   // GBK_TO_UNICODE[30877] := 16#502D;
   // GBK_TO_UNICODE[30878] := 16#D9C2;
   // GBK_TO_UNICODE[30879] := 16#4FFE;
   // GBK_TO_UNICODE[30880] := 16#D9C3;
   // GBK_TO_UNICODE[30881] := 16#501C;
   // GBK_TO_UNICODE[30882] := 16#D9C4;
   // GBK_TO_UNICODE[30883] := 16#500C;
   // GBK_TO_UNICODE[30884] := 16#D9C5;
   // GBK_TO_UNICODE[30885] := 16#5025;
   // GBK_TO_UNICODE[30886] := 16#D9C6;
   // GBK_TO_UNICODE[30887] := 16#5028;
   // GBK_TO_UNICODE[30888] := 16#D9C7;
   // GBK_TO_UNICODE[30889] := 16#507E;
   // GBK_TO_UNICODE[30890] := 16#D9C8;
   // GBK_TO_UNICODE[30891] := 16#5043;
   // GBK_TO_UNICODE[30892] := 16#D9C9;
   // GBK_TO_UNICODE[30893] := 16#5055;
   // GBK_TO_UNICODE[30894] := 16#D9CA;
   // GBK_TO_UNICODE[30895] := 16#5048;
   // GBK_TO_UNICODE[30896] := 16#D9CB;
   // GBK_TO_UNICODE[30897] := 16#504E;
   // GBK_TO_UNICODE[30898] := 16#D9CC;
   // GBK_TO_UNICODE[30899] := 16#506C;
   // GBK_TO_UNICODE[30900] := 16#D9CD;
   // GBK_TO_UNICODE[30901] := 16#507B;
   // GBK_TO_UNICODE[30902] := 16#D9CE;
   // GBK_TO_UNICODE[30903] := 16#50A5;
   // GBK_TO_UNICODE[30904] := 16#D9CF;
   // GBK_TO_UNICODE[30905] := 16#50A7;
   // GBK_TO_UNICODE[30906] := 16#D9D0;
   // GBK_TO_UNICODE[30907] := 16#50A9;
   // GBK_TO_UNICODE[30908] := 16#D9D1;
   // GBK_TO_UNICODE[30909] := 16#50BA;
   // GBK_TO_UNICODE[30910] := 16#D9D2;
   // GBK_TO_UNICODE[30911] := 16#50D6;
   // GBK_TO_UNICODE[30912] := 16#D9D3;
   // GBK_TO_UNICODE[30913] := 16#5106;
   // GBK_TO_UNICODE[30914] := 16#D9D4;
   // GBK_TO_UNICODE[30915] := 16#50ED;
   // GBK_TO_UNICODE[30916] := 16#D9D5;
   // GBK_TO_UNICODE[30917] := 16#50EC;
   // GBK_TO_UNICODE[30918] := 16#D9D6;
   // GBK_TO_UNICODE[30919] := 16#50E6;
   // GBK_TO_UNICODE[30920] := 16#D9D7;
   // GBK_TO_UNICODE[30921] := 16#50EE;
   // GBK_TO_UNICODE[30922] := 16#D9D8;
   // GBK_TO_UNICODE[30923] := 16#5107;
   // GBK_TO_UNICODE[30924] := 16#D9D9;
   // GBK_TO_UNICODE[30925] := 16#510B;
   // GBK_TO_UNICODE[30926] := 16#D9DA;
   // GBK_TO_UNICODE[30927] := 16#4EDD;
   // GBK_TO_UNICODE[30928] := 16#D9DB;
   // GBK_TO_UNICODE[30929] := 16#6C3D;
   // GBK_TO_UNICODE[30930] := 16#D9DC;
   // GBK_TO_UNICODE[30931] := 16#4F58;
   // GBK_TO_UNICODE[30932] := 16#D9DD;
   // GBK_TO_UNICODE[30933] := 16#4F65;
   // GBK_TO_UNICODE[30934] := 16#D9DE;
   // GBK_TO_UNICODE[30935] := 16#4FCE;
   // GBK_TO_UNICODE[30936] := 16#D9DF;
   // GBK_TO_UNICODE[30937] := 16#9FA0;
   // GBK_TO_UNICODE[30938] := 16#D9E0;
   // GBK_TO_UNICODE[30939] := 16#6C46;
   // GBK_TO_UNICODE[30940] := 16#D9E1;
   // GBK_TO_UNICODE[30941] := 16#7C74;
   // GBK_TO_UNICODE[30942] := 16#D9E2;
   // GBK_TO_UNICODE[30943] := 16#516E;
   // GBK_TO_UNICODE[30944] := 16#D9E3;
   // GBK_TO_UNICODE[30945] := 16#5DFD;
   // GBK_TO_UNICODE[30946] := 16#D9E4;
   // GBK_TO_UNICODE[30947] := 16#9EC9;
   // GBK_TO_UNICODE[30948] := 16#D9E5;
   // GBK_TO_UNICODE[30949] := 16#9998;
   // GBK_TO_UNICODE[30950] := 16#D9E6;
   // GBK_TO_UNICODE[30951] := 16#5181;
   // GBK_TO_UNICODE[30952] := 16#D9E7;
   // GBK_TO_UNICODE[30953] := 16#5914;
   // GBK_TO_UNICODE[30954] := 16#D9E8;
   // GBK_TO_UNICODE[30955] := 16#52F9;
   // GBK_TO_UNICODE[30956] := 16#D9E9;
   // GBK_TO_UNICODE[30957] := 16#530D;
   // GBK_TO_UNICODE[30958] := 16#D9EA;
   // GBK_TO_UNICODE[30959] := 16#8A07;
   // GBK_TO_UNICODE[30960] := 16#D9EB;
   // GBK_TO_UNICODE[30961] := 16#5310;
   // GBK_TO_UNICODE[30962] := 16#D9EC;
   // GBK_TO_UNICODE[30963] := 16#51EB;
   // GBK_TO_UNICODE[30964] := 16#D9ED;
   // GBK_TO_UNICODE[30965] := 16#5919;
   // GBK_TO_UNICODE[30966] := 16#D9EE;
   // GBK_TO_UNICODE[30967] := 16#5155;
   // GBK_TO_UNICODE[30968] := 16#D9EF;
   // GBK_TO_UNICODE[30969] := 16#4EA0;
   // GBK_TO_UNICODE[30970] := 16#D9F0;
   // GBK_TO_UNICODE[30971] := 16#5156;
   // GBK_TO_UNICODE[30972] := 16#D9F1;
   // GBK_TO_UNICODE[30973] := 16#4EB3;
   // GBK_TO_UNICODE[30974] := 16#D9F2;
   // GBK_TO_UNICODE[30975] := 16#886E;
   // GBK_TO_UNICODE[30976] := 16#D9F3;
   // GBK_TO_UNICODE[30977] := 16#88A4;
   // GBK_TO_UNICODE[30978] := 16#D9F4;
   // GBK_TO_UNICODE[30979] := 16#4EB5;
   // GBK_TO_UNICODE[30980] := 16#D9F5;
   // GBK_TO_UNICODE[30981] := 16#8114;
   // GBK_TO_UNICODE[30982] := 16#D9F6;
   // GBK_TO_UNICODE[30983] := 16#88D2;
   // GBK_TO_UNICODE[30984] := 16#D9F7;
   // GBK_TO_UNICODE[30985] := 16#7980;
   // GBK_TO_UNICODE[30986] := 16#D9F8;
   // GBK_TO_UNICODE[30987] := 16#5B34;
   // GBK_TO_UNICODE[30988] := 16#D9F9;
   // GBK_TO_UNICODE[30989] := 16#8803;
   // GBK_TO_UNICODE[30990] := 16#D9FA;
   // GBK_TO_UNICODE[30991] := 16#7FB8;
   // GBK_TO_UNICODE[30992] := 16#D9FB;
   // GBK_TO_UNICODE[30993] := 16#51AB;
   // GBK_TO_UNICODE[30994] := 16#D9FC;
   // GBK_TO_UNICODE[30995] := 16#51B1;
   // GBK_TO_UNICODE[30996] := 16#D9FD;
   // GBK_TO_UNICODE[30997] := 16#51BD;
   // GBK_TO_UNICODE[30998] := 16#D9FE;
   // GBK_TO_UNICODE[30999] := 16#51BC;
   // GBK_TO_UNICODE[31000] := 16#DA40;
   // GBK_TO_UNICODE[31001] := 16#8D0E;
   // GBK_TO_UNICODE[31002] := 16#DA41;
   // GBK_TO_UNICODE[31003] := 16#8D0F;
   // GBK_TO_UNICODE[31004] := 16#DA42;
   // GBK_TO_UNICODE[31005] := 16#8D10;
   // GBK_TO_UNICODE[31006] := 16#DA43;
   // GBK_TO_UNICODE[31007] := 16#8D11;
   // GBK_TO_UNICODE[31008] := 16#DA44;
   // GBK_TO_UNICODE[31009] := 16#8D12;
   // GBK_TO_UNICODE[31010] := 16#DA45;
   // GBK_TO_UNICODE[31011] := 16#8D13;
   // GBK_TO_UNICODE[31012] := 16#DA46;
   // GBK_TO_UNICODE[31013] := 16#8D14;
   // GBK_TO_UNICODE[31014] := 16#DA47;
   // GBK_TO_UNICODE[31015] := 16#8D15;
   // GBK_TO_UNICODE[31016] := 16#DA48;
   // GBK_TO_UNICODE[31017] := 16#8D16;
   // GBK_TO_UNICODE[31018] := 16#DA49;
   // GBK_TO_UNICODE[31019] := 16#8D17;
   // GBK_TO_UNICODE[31020] := 16#DA4A;
   // GBK_TO_UNICODE[31021] := 16#8D18;
   // GBK_TO_UNICODE[31022] := 16#DA4B;
   // GBK_TO_UNICODE[31023] := 16#8D19;
   // GBK_TO_UNICODE[31024] := 16#DA4C;
   // GBK_TO_UNICODE[31025] := 16#8D1A;
   // GBK_TO_UNICODE[31026] := 16#DA4D;
   // GBK_TO_UNICODE[31027] := 16#8D1B;
   // GBK_TO_UNICODE[31028] := 16#DA4E;
   // GBK_TO_UNICODE[31029] := 16#8D1C;
   // GBK_TO_UNICODE[31030] := 16#DA4F;
   // GBK_TO_UNICODE[31031] := 16#8D20;
   // GBK_TO_UNICODE[31032] := 16#DA50;
   // GBK_TO_UNICODE[31033] := 16#8D51;
   // GBK_TO_UNICODE[31034] := 16#DA51;
   // GBK_TO_UNICODE[31035] := 16#8D52;
   // GBK_TO_UNICODE[31036] := 16#DA52;
   // GBK_TO_UNICODE[31037] := 16#8D57;
   // GBK_TO_UNICODE[31038] := 16#DA53;
   // GBK_TO_UNICODE[31039] := 16#8D5F;
   // GBK_TO_UNICODE[31040] := 16#DA54;
   // GBK_TO_UNICODE[31041] := 16#8D65;
   // GBK_TO_UNICODE[31042] := 16#DA55;
   // GBK_TO_UNICODE[31043] := 16#8D68;
   // GBK_TO_UNICODE[31044] := 16#DA56;
   // GBK_TO_UNICODE[31045] := 16#8D69;
   // GBK_TO_UNICODE[31046] := 16#DA57;
   // GBK_TO_UNICODE[31047] := 16#8D6A;
   // GBK_TO_UNICODE[31048] := 16#DA58;
   // GBK_TO_UNICODE[31049] := 16#8D6C;
   // GBK_TO_UNICODE[31050] := 16#DA59;
   // GBK_TO_UNICODE[31051] := 16#8D6E;
   // GBK_TO_UNICODE[31052] := 16#DA5A;
   // GBK_TO_UNICODE[31053] := 16#8D6F;
   // GBK_TO_UNICODE[31054] := 16#DA5B;
   // GBK_TO_UNICODE[31055] := 16#8D71;
   // GBK_TO_UNICODE[31056] := 16#DA5C;
   // GBK_TO_UNICODE[31057] := 16#8D72;
   // GBK_TO_UNICODE[31058] := 16#DA5D;
   // GBK_TO_UNICODE[31059] := 16#8D78;
   // GBK_TO_UNICODE[31060] := 16#DA5E;
   // GBK_TO_UNICODE[31061] := 16#8D79;
   // GBK_TO_UNICODE[31062] := 16#DA5F;
   // GBK_TO_UNICODE[31063] := 16#8D7A;
   // GBK_TO_UNICODE[31064] := 16#DA60;
   // GBK_TO_UNICODE[31065] := 16#8D7B;
   // GBK_TO_UNICODE[31066] := 16#DA61;
   // GBK_TO_UNICODE[31067] := 16#8D7C;
   // GBK_TO_UNICODE[31068] := 16#DA62;
   // GBK_TO_UNICODE[31069] := 16#8D7D;
   // GBK_TO_UNICODE[31070] := 16#DA63;
   // GBK_TO_UNICODE[31071] := 16#8D7E;
   // GBK_TO_UNICODE[31072] := 16#DA64;
   // GBK_TO_UNICODE[31073] := 16#8D7F;
   // GBK_TO_UNICODE[31074] := 16#DA65;
   // GBK_TO_UNICODE[31075] := 16#8D80;
   // GBK_TO_UNICODE[31076] := 16#DA66;
   // GBK_TO_UNICODE[31077] := 16#8D82;
   // GBK_TO_UNICODE[31078] := 16#DA67;
   // GBK_TO_UNICODE[31079] := 16#8D83;
   // GBK_TO_UNICODE[31080] := 16#DA68;
   // GBK_TO_UNICODE[31081] := 16#8D86;
   // GBK_TO_UNICODE[31082] := 16#DA69;
   // GBK_TO_UNICODE[31083] := 16#8D87;
   // GBK_TO_UNICODE[31084] := 16#DA6A;
   // GBK_TO_UNICODE[31085] := 16#8D88;
   // GBK_TO_UNICODE[31086] := 16#DA6B;
   // GBK_TO_UNICODE[31087] := 16#8D89;
   // GBK_TO_UNICODE[31088] := 16#DA6C;
   // GBK_TO_UNICODE[31089] := 16#8D8C;
   // GBK_TO_UNICODE[31090] := 16#DA6D;
   // GBK_TO_UNICODE[31091] := 16#8D8D;
   // GBK_TO_UNICODE[31092] := 16#DA6E;
   // GBK_TO_UNICODE[31093] := 16#8D8E;
   // GBK_TO_UNICODE[31094] := 16#DA6F;
   // GBK_TO_UNICODE[31095] := 16#8D8F;
   // GBK_TO_UNICODE[31096] := 16#DA70;
   // GBK_TO_UNICODE[31097] := 16#8D90;
   // GBK_TO_UNICODE[31098] := 16#DA71;
   // GBK_TO_UNICODE[31099] := 16#8D92;
   // GBK_TO_UNICODE[31100] := 16#DA72;
   // GBK_TO_UNICODE[31101] := 16#8D93;
   // GBK_TO_UNICODE[31102] := 16#DA73;
   // GBK_TO_UNICODE[31103] := 16#8D95;
   // GBK_TO_UNICODE[31104] := 16#DA74;
   // GBK_TO_UNICODE[31105] := 16#8D96;
   // GBK_TO_UNICODE[31106] := 16#DA75;
   // GBK_TO_UNICODE[31107] := 16#8D97;
   // GBK_TO_UNICODE[31108] := 16#DA76;
   // GBK_TO_UNICODE[31109] := 16#8D98;
   // GBK_TO_UNICODE[31110] := 16#DA77;
   // GBK_TO_UNICODE[31111] := 16#8D99;
   // GBK_TO_UNICODE[31112] := 16#DA78;
   // GBK_TO_UNICODE[31113] := 16#8D9A;
   // GBK_TO_UNICODE[31114] := 16#DA79;
   // GBK_TO_UNICODE[31115] := 16#8D9B;
   // GBK_TO_UNICODE[31116] := 16#DA7A;
   // GBK_TO_UNICODE[31117] := 16#8D9C;
   // GBK_TO_UNICODE[31118] := 16#DA7B;
   // GBK_TO_UNICODE[31119] := 16#8D9D;
   // GBK_TO_UNICODE[31120] := 16#DA7C;
   // GBK_TO_UNICODE[31121] := 16#8D9E;
   // GBK_TO_UNICODE[31122] := 16#DA7D;
   // GBK_TO_UNICODE[31123] := 16#8DA0;
   // GBK_TO_UNICODE[31124] := 16#DA7E;
   // GBK_TO_UNICODE[31125] := 16#8DA1;
   // GBK_TO_UNICODE[31126] := 16#DA80;
   // GBK_TO_UNICODE[31127] := 16#8DA2;
   // GBK_TO_UNICODE[31128] := 16#DA81;
   // GBK_TO_UNICODE[31129] := 16#8DA4;
   // GBK_TO_UNICODE[31130] := 16#DA82;
   // GBK_TO_UNICODE[31131] := 16#8DA5;
   // GBK_TO_UNICODE[31132] := 16#DA83;
   // GBK_TO_UNICODE[31133] := 16#8DA6;
   // GBK_TO_UNICODE[31134] := 16#DA84;
   // GBK_TO_UNICODE[31135] := 16#8DA7;
   // GBK_TO_UNICODE[31136] := 16#DA85;
   // GBK_TO_UNICODE[31137] := 16#8DA8;
   // GBK_TO_UNICODE[31138] := 16#DA86;
   // GBK_TO_UNICODE[31139] := 16#8DA9;
   // GBK_TO_UNICODE[31140] := 16#DA87;
   // GBK_TO_UNICODE[31141] := 16#8DAA;
   // GBK_TO_UNICODE[31142] := 16#DA88;
   // GBK_TO_UNICODE[31143] := 16#8DAB;
   // GBK_TO_UNICODE[31144] := 16#DA89;
   // GBK_TO_UNICODE[31145] := 16#8DAC;
   // GBK_TO_UNICODE[31146] := 16#DA8A;
   // GBK_TO_UNICODE[31147] := 16#8DAD;
   // GBK_TO_UNICODE[31148] := 16#DA8B;
   // GBK_TO_UNICODE[31149] := 16#8DAE;
   // GBK_TO_UNICODE[31150] := 16#DA8C;
   // GBK_TO_UNICODE[31151] := 16#8DAF;
   // GBK_TO_UNICODE[31152] := 16#DA8D;
   // GBK_TO_UNICODE[31153] := 16#8DB0;
   // GBK_TO_UNICODE[31154] := 16#DA8E;
   // GBK_TO_UNICODE[31155] := 16#8DB2;
   // GBK_TO_UNICODE[31156] := 16#DA8F;
   // GBK_TO_UNICODE[31157] := 16#8DB6;
   // GBK_TO_UNICODE[31158] := 16#DA90;
   // GBK_TO_UNICODE[31159] := 16#8DB7;
   // GBK_TO_UNICODE[31160] := 16#DA91;
   // GBK_TO_UNICODE[31161] := 16#8DB9;
   // GBK_TO_UNICODE[31162] := 16#DA92;
   // GBK_TO_UNICODE[31163] := 16#8DBB;
   // GBK_TO_UNICODE[31164] := 16#DA93;
   // GBK_TO_UNICODE[31165] := 16#8DBD;
   // GBK_TO_UNICODE[31166] := 16#DA94;
   // GBK_TO_UNICODE[31167] := 16#8DC0;
   // GBK_TO_UNICODE[31168] := 16#DA95;
   // GBK_TO_UNICODE[31169] := 16#8DC1;
   // GBK_TO_UNICODE[31170] := 16#DA96;
   // GBK_TO_UNICODE[31171] := 16#8DC2;
   // GBK_TO_UNICODE[31172] := 16#DA97;
   // GBK_TO_UNICODE[31173] := 16#8DC5;
   // GBK_TO_UNICODE[31174] := 16#DA98;
   // GBK_TO_UNICODE[31175] := 16#8DC7;
   // GBK_TO_UNICODE[31176] := 16#DA99;
   // GBK_TO_UNICODE[31177] := 16#8DC8;
   // GBK_TO_UNICODE[31178] := 16#DA9A;
   // GBK_TO_UNICODE[31179] := 16#8DC9;
   // GBK_TO_UNICODE[31180] := 16#DA9B;
   // GBK_TO_UNICODE[31181] := 16#8DCA;
   // GBK_TO_UNICODE[31182] := 16#DA9C;
   // GBK_TO_UNICODE[31183] := 16#8DCD;
   // GBK_TO_UNICODE[31184] := 16#DA9D;
   // GBK_TO_UNICODE[31185] := 16#8DD0;
   // GBK_TO_UNICODE[31186] := 16#DA9E;
   // GBK_TO_UNICODE[31187] := 16#8DD2;
   // GBK_TO_UNICODE[31188] := 16#DA9F;
   // GBK_TO_UNICODE[31189] := 16#8DD3;
   // GBK_TO_UNICODE[31190] := 16#DAA0;
   // GBK_TO_UNICODE[31191] := 16#8DD4;
   // GBK_TO_UNICODE[31192] := 16#DAA1;
   // GBK_TO_UNICODE[31193] := 16#51C7;
   // GBK_TO_UNICODE[31194] := 16#DAA2;
   // GBK_TO_UNICODE[31195] := 16#5196;
   // GBK_TO_UNICODE[31196] := 16#DAA3;
   // GBK_TO_UNICODE[31197] := 16#51A2;
   // GBK_TO_UNICODE[31198] := 16#DAA4;
   // GBK_TO_UNICODE[31199] := 16#51A5;
   // GBK_TO_UNICODE[31200] := 16#DAA5;
   // GBK_TO_UNICODE[31201] := 16#8BA0;
   // GBK_TO_UNICODE[31202] := 16#DAA6;
   // GBK_TO_UNICODE[31203] := 16#8BA6;
   // GBK_TO_UNICODE[31204] := 16#DAA7;
   // GBK_TO_UNICODE[31205] := 16#8BA7;
   // GBK_TO_UNICODE[31206] := 16#DAA8;
   // GBK_TO_UNICODE[31207] := 16#8BAA;
   // GBK_TO_UNICODE[31208] := 16#DAA9;
   // GBK_TO_UNICODE[31209] := 16#8BB4;
   // GBK_TO_UNICODE[31210] := 16#DAAA;
   // GBK_TO_UNICODE[31211] := 16#8BB5;
   // GBK_TO_UNICODE[31212] := 16#DAAB;
   // GBK_TO_UNICODE[31213] := 16#8BB7;
   // GBK_TO_UNICODE[31214] := 16#DAAC;
   // GBK_TO_UNICODE[31215] := 16#8BC2;
   // GBK_TO_UNICODE[31216] := 16#DAAD;
   // GBK_TO_UNICODE[31217] := 16#8BC3;
   // GBK_TO_UNICODE[31218] := 16#DAAE;
   // GBK_TO_UNICODE[31219] := 16#8BCB;
   // GBK_TO_UNICODE[31220] := 16#DAAF;
   // GBK_TO_UNICODE[31221] := 16#8BCF;
   // GBK_TO_UNICODE[31222] := 16#DAB0;
   // GBK_TO_UNICODE[31223] := 16#8BCE;
   // GBK_TO_UNICODE[31224] := 16#DAB1;
   // GBK_TO_UNICODE[31225] := 16#8BD2;
   // GBK_TO_UNICODE[31226] := 16#DAB2;
   // GBK_TO_UNICODE[31227] := 16#8BD3;
   // GBK_TO_UNICODE[31228] := 16#DAB3;
   // GBK_TO_UNICODE[31229] := 16#8BD4;
   // GBK_TO_UNICODE[31230] := 16#DAB4;
   // GBK_TO_UNICODE[31231] := 16#8BD6;
   // GBK_TO_UNICODE[31232] := 16#DAB5;
   // GBK_TO_UNICODE[31233] := 16#8BD8;
   // GBK_TO_UNICODE[31234] := 16#DAB6;
   // GBK_TO_UNICODE[31235] := 16#8BD9;
   // GBK_TO_UNICODE[31236] := 16#DAB7;
   // GBK_TO_UNICODE[31237] := 16#8BDC;
   // GBK_TO_UNICODE[31238] := 16#DAB8;
   // GBK_TO_UNICODE[31239] := 16#8BDF;
   // GBK_TO_UNICODE[31240] := 16#DAB9;
   // GBK_TO_UNICODE[31241] := 16#8BE0;
   // GBK_TO_UNICODE[31242] := 16#DABA;
   // GBK_TO_UNICODE[31243] := 16#8BE4;
   // GBK_TO_UNICODE[31244] := 16#DABB;
   // GBK_TO_UNICODE[31245] := 16#8BE8;
   // GBK_TO_UNICODE[31246] := 16#DABC;
   // GBK_TO_UNICODE[31247] := 16#8BE9;
   // GBK_TO_UNICODE[31248] := 16#DABD;
   // GBK_TO_UNICODE[31249] := 16#8BEE;
   // GBK_TO_UNICODE[31250] := 16#DABE;
   // GBK_TO_UNICODE[31251] := 16#8BF0;
   // GBK_TO_UNICODE[31252] := 16#DABF;
   // GBK_TO_UNICODE[31253] := 16#8BF3;
   // GBK_TO_UNICODE[31254] := 16#DAC0;
   // GBK_TO_UNICODE[31255] := 16#8BF6;
   // GBK_TO_UNICODE[31256] := 16#DAC1;
   // GBK_TO_UNICODE[31257] := 16#8BF9;
   // GBK_TO_UNICODE[31258] := 16#DAC2;
   // GBK_TO_UNICODE[31259] := 16#8BFC;
   // GBK_TO_UNICODE[31260] := 16#DAC3;
   // GBK_TO_UNICODE[31261] := 16#8BFF;
   // GBK_TO_UNICODE[31262] := 16#DAC4;
   // GBK_TO_UNICODE[31263] := 16#8C00;
   // GBK_TO_UNICODE[31264] := 16#DAC5;
   // GBK_TO_UNICODE[31265] := 16#8C02;
   // GBK_TO_UNICODE[31266] := 16#DAC6;
   // GBK_TO_UNICODE[31267] := 16#8C04;
   // GBK_TO_UNICODE[31268] := 16#DAC7;
   // GBK_TO_UNICODE[31269] := 16#8C07;
   // GBK_TO_UNICODE[31270] := 16#DAC8;
   // GBK_TO_UNICODE[31271] := 16#8C0C;
   // GBK_TO_UNICODE[31272] := 16#DAC9;
   // GBK_TO_UNICODE[31273] := 16#8C0F;
   // GBK_TO_UNICODE[31274] := 16#DACA;
   // GBK_TO_UNICODE[31275] := 16#8C11;
   // GBK_TO_UNICODE[31276] := 16#DACB;
   // GBK_TO_UNICODE[31277] := 16#8C12;
   // GBK_TO_UNICODE[31278] := 16#DACC;
   // GBK_TO_UNICODE[31279] := 16#8C14;
   // GBK_TO_UNICODE[31280] := 16#DACD;
   // GBK_TO_UNICODE[31281] := 16#8C15;
   // GBK_TO_UNICODE[31282] := 16#DACE;
   // GBK_TO_UNICODE[31283] := 16#8C16;
   // GBK_TO_UNICODE[31284] := 16#DACF;
   // GBK_TO_UNICODE[31285] := 16#8C19;
   // GBK_TO_UNICODE[31286] := 16#DAD0;
   // GBK_TO_UNICODE[31287] := 16#8C1B;
   // GBK_TO_UNICODE[31288] := 16#DAD1;
   // GBK_TO_UNICODE[31289] := 16#8C18;
   // GBK_TO_UNICODE[31290] := 16#DAD2;
   // GBK_TO_UNICODE[31291] := 16#8C1D;
   // GBK_TO_UNICODE[31292] := 16#DAD3;
   // GBK_TO_UNICODE[31293] := 16#8C1F;
   // GBK_TO_UNICODE[31294] := 16#DAD4;
   // GBK_TO_UNICODE[31295] := 16#8C20;
   // GBK_TO_UNICODE[31296] := 16#DAD5;
   // GBK_TO_UNICODE[31297] := 16#8C21;
   // GBK_TO_UNICODE[31298] := 16#DAD6;
   // GBK_TO_UNICODE[31299] := 16#8C25;
   // GBK_TO_UNICODE[31300] := 16#DAD7;
   // GBK_TO_UNICODE[31301] := 16#8C27;
   // GBK_TO_UNICODE[31302] := 16#DAD8;
   // GBK_TO_UNICODE[31303] := 16#8C2A;
   // GBK_TO_UNICODE[31304] := 16#DAD9;
   // GBK_TO_UNICODE[31305] := 16#8C2B;
   // GBK_TO_UNICODE[31306] := 16#DADA;
   // GBK_TO_UNICODE[31307] := 16#8C2E;
   // GBK_TO_UNICODE[31308] := 16#DADB;
   // GBK_TO_UNICODE[31309] := 16#8C2F;
   // GBK_TO_UNICODE[31310] := 16#DADC;
   // GBK_TO_UNICODE[31311] := 16#8C32;
   // GBK_TO_UNICODE[31312] := 16#DADD;
   // GBK_TO_UNICODE[31313] := 16#8C33;
   // GBK_TO_UNICODE[31314] := 16#DADE;
   // GBK_TO_UNICODE[31315] := 16#8C35;
   // GBK_TO_UNICODE[31316] := 16#DADF;
   // GBK_TO_UNICODE[31317] := 16#8C36;
   // GBK_TO_UNICODE[31318] := 16#DAE0;
   // GBK_TO_UNICODE[31319] := 16#5369;
   // GBK_TO_UNICODE[31320] := 16#DAE1;
   // GBK_TO_UNICODE[31321] := 16#537A;
   // GBK_TO_UNICODE[31322] := 16#DAE2;
   // GBK_TO_UNICODE[31323] := 16#961D;
   // GBK_TO_UNICODE[31324] := 16#DAE3;
   // GBK_TO_UNICODE[31325] := 16#9622;
   // GBK_TO_UNICODE[31326] := 16#DAE4;
   // GBK_TO_UNICODE[31327] := 16#9621;
   // GBK_TO_UNICODE[31328] := 16#DAE5;
   // GBK_TO_UNICODE[31329] := 16#9631;
   // GBK_TO_UNICODE[31330] := 16#DAE6;
   // GBK_TO_UNICODE[31331] := 16#962A;
   // GBK_TO_UNICODE[31332] := 16#DAE7;
   // GBK_TO_UNICODE[31333] := 16#963D;
   // GBK_TO_UNICODE[31334] := 16#DAE8;
   // GBK_TO_UNICODE[31335] := 16#963C;
   // GBK_TO_UNICODE[31336] := 16#DAE9;
   // GBK_TO_UNICODE[31337] := 16#9642;
   // GBK_TO_UNICODE[31338] := 16#DAEA;
   // GBK_TO_UNICODE[31339] := 16#9649;
   // GBK_TO_UNICODE[31340] := 16#DAEB;
   // GBK_TO_UNICODE[31341] := 16#9654;
   // GBK_TO_UNICODE[31342] := 16#DAEC;
   // GBK_TO_UNICODE[31343] := 16#965F;
   // GBK_TO_UNICODE[31344] := 16#DAED;
   // GBK_TO_UNICODE[31345] := 16#9667;
   // GBK_TO_UNICODE[31346] := 16#DAEE;
   // GBK_TO_UNICODE[31347] := 16#966C;
   // GBK_TO_UNICODE[31348] := 16#DAEF;
   // GBK_TO_UNICODE[31349] := 16#9672;
   // GBK_TO_UNICODE[31350] := 16#DAF0;
   // GBK_TO_UNICODE[31351] := 16#9674;
   // GBK_TO_UNICODE[31352] := 16#DAF1;
   // GBK_TO_UNICODE[31353] := 16#9688;
   // GBK_TO_UNICODE[31354] := 16#DAF2;
   // GBK_TO_UNICODE[31355] := 16#968D;
   // GBK_TO_UNICODE[31356] := 16#DAF3;
   // GBK_TO_UNICODE[31357] := 16#9697;
   // GBK_TO_UNICODE[31358] := 16#DAF4;
   // GBK_TO_UNICODE[31359] := 16#96B0;
   // GBK_TO_UNICODE[31360] := 16#DAF5;
   // GBK_TO_UNICODE[31361] := 16#9097;
   // GBK_TO_UNICODE[31362] := 16#DAF6;
   // GBK_TO_UNICODE[31363] := 16#909B;
   // GBK_TO_UNICODE[31364] := 16#DAF7;
   // GBK_TO_UNICODE[31365] := 16#909D;
   // GBK_TO_UNICODE[31366] := 16#DAF8;
   // GBK_TO_UNICODE[31367] := 16#9099;
   // GBK_TO_UNICODE[31368] := 16#DAF9;
   // GBK_TO_UNICODE[31369] := 16#90AC;
   // GBK_TO_UNICODE[31370] := 16#DAFA;
   // GBK_TO_UNICODE[31371] := 16#90A1;
   // GBK_TO_UNICODE[31372] := 16#DAFB;
   // GBK_TO_UNICODE[31373] := 16#90B4;
   // GBK_TO_UNICODE[31374] := 16#DAFC;
   // GBK_TO_UNICODE[31375] := 16#90B3;
   // GBK_TO_UNICODE[31376] := 16#DAFD;
   // GBK_TO_UNICODE[31377] := 16#90B6;
   // GBK_TO_UNICODE[31378] := 16#DAFE;
   // GBK_TO_UNICODE[31379] := 16#90BA;
   // GBK_TO_UNICODE[31380] := 16#DB40;
   // GBK_TO_UNICODE[31381] := 16#8DD5;
   // GBK_TO_UNICODE[31382] := 16#DB41;
   // GBK_TO_UNICODE[31383] := 16#8DD8;
   // GBK_TO_UNICODE[31384] := 16#DB42;
   // GBK_TO_UNICODE[31385] := 16#8DD9;
   // GBK_TO_UNICODE[31386] := 16#DB43;
   // GBK_TO_UNICODE[31387] := 16#8DDC;
   // GBK_TO_UNICODE[31388] := 16#DB44;
   // GBK_TO_UNICODE[31389] := 16#8DE0;
   // GBK_TO_UNICODE[31390] := 16#DB45;
   // GBK_TO_UNICODE[31391] := 16#8DE1;
   // GBK_TO_UNICODE[31392] := 16#DB46;
   // GBK_TO_UNICODE[31393] := 16#8DE2;
   // GBK_TO_UNICODE[31394] := 16#DB47;
   // GBK_TO_UNICODE[31395] := 16#8DE5;
   // GBK_TO_UNICODE[31396] := 16#DB48;
   // GBK_TO_UNICODE[31397] := 16#8DE6;
   // GBK_TO_UNICODE[31398] := 16#DB49;
   // GBK_TO_UNICODE[31399] := 16#8DE7;
   // GBK_TO_UNICODE[31400] := 16#DB4A;
   // GBK_TO_UNICODE[31401] := 16#8DE9;
   // GBK_TO_UNICODE[31402] := 16#DB4B;
   // GBK_TO_UNICODE[31403] := 16#8DED;
   // GBK_TO_UNICODE[31404] := 16#DB4C;
   // GBK_TO_UNICODE[31405] := 16#8DEE;
   // GBK_TO_UNICODE[31406] := 16#DB4D;
   // GBK_TO_UNICODE[31407] := 16#8DF0;
   // GBK_TO_UNICODE[31408] := 16#DB4E;
   // GBK_TO_UNICODE[31409] := 16#8DF1;
   // GBK_TO_UNICODE[31410] := 16#DB4F;
   // GBK_TO_UNICODE[31411] := 16#8DF2;
   // GBK_TO_UNICODE[31412] := 16#DB50;
   // GBK_TO_UNICODE[31413] := 16#8DF4;
   // GBK_TO_UNICODE[31414] := 16#DB51;
   // GBK_TO_UNICODE[31415] := 16#8DF6;
   // GBK_TO_UNICODE[31416] := 16#DB52;
   // GBK_TO_UNICODE[31417] := 16#8DFC;
   // GBK_TO_UNICODE[31418] := 16#DB53;
   // GBK_TO_UNICODE[31419] := 16#8DFE;
   // GBK_TO_UNICODE[31420] := 16#DB54;
   // GBK_TO_UNICODE[31421] := 16#8DFF;
   // GBK_TO_UNICODE[31422] := 16#DB55;
   // GBK_TO_UNICODE[31423] := 16#8E00;
   // GBK_TO_UNICODE[31424] := 16#DB56;
   // GBK_TO_UNICODE[31425] := 16#8E01;
   // GBK_TO_UNICODE[31426] := 16#DB57;
   // GBK_TO_UNICODE[31427] := 16#8E02;
   // GBK_TO_UNICODE[31428] := 16#DB58;
   // GBK_TO_UNICODE[31429] := 16#8E03;
   // GBK_TO_UNICODE[31430] := 16#DB59;
   // GBK_TO_UNICODE[31431] := 16#8E04;
   // GBK_TO_UNICODE[31432] := 16#DB5A;
   // GBK_TO_UNICODE[31433] := 16#8E06;
   // GBK_TO_UNICODE[31434] := 16#DB5B;
   // GBK_TO_UNICODE[31435] := 16#8E07;
   // GBK_TO_UNICODE[31436] := 16#DB5C;
   // GBK_TO_UNICODE[31437] := 16#8E08;
   // GBK_TO_UNICODE[31438] := 16#DB5D;
   // GBK_TO_UNICODE[31439] := 16#8E0B;
   // GBK_TO_UNICODE[31440] := 16#DB5E;
   // GBK_TO_UNICODE[31441] := 16#8E0D;
   // GBK_TO_UNICODE[31442] := 16#DB5F;
   // GBK_TO_UNICODE[31443] := 16#8E0E;
   // GBK_TO_UNICODE[31444] := 16#DB60;
   // GBK_TO_UNICODE[31445] := 16#8E10;
   // GBK_TO_UNICODE[31446] := 16#DB61;
   // GBK_TO_UNICODE[31447] := 16#8E11;
   // GBK_TO_UNICODE[31448] := 16#DB62;
   // GBK_TO_UNICODE[31449] := 16#8E12;
   // GBK_TO_UNICODE[31450] := 16#DB63;
   // GBK_TO_UNICODE[31451] := 16#8E13;
   // GBK_TO_UNICODE[31452] := 16#DB64;
   // GBK_TO_UNICODE[31453] := 16#8E15;
   // GBK_TO_UNICODE[31454] := 16#DB65;
   // GBK_TO_UNICODE[31455] := 16#8E16;
   // GBK_TO_UNICODE[31456] := 16#DB66;
   // GBK_TO_UNICODE[31457] := 16#8E17;
   // GBK_TO_UNICODE[31458] := 16#DB67;
   // GBK_TO_UNICODE[31459] := 16#8E18;
   // GBK_TO_UNICODE[31460] := 16#DB68;
   // GBK_TO_UNICODE[31461] := 16#8E19;
   // GBK_TO_UNICODE[31462] := 16#DB69;
   // GBK_TO_UNICODE[31463] := 16#8E1A;
   // GBK_TO_UNICODE[31464] := 16#DB6A;
   // GBK_TO_UNICODE[31465] := 16#8E1B;
   // GBK_TO_UNICODE[31466] := 16#DB6B;
   // GBK_TO_UNICODE[31467] := 16#8E1C;
   // GBK_TO_UNICODE[31468] := 16#DB6C;
   // GBK_TO_UNICODE[31469] := 16#8E20;
   // GBK_TO_UNICODE[31470] := 16#DB6D;
   // GBK_TO_UNICODE[31471] := 16#8E21;
   // GBK_TO_UNICODE[31472] := 16#DB6E;
   // GBK_TO_UNICODE[31473] := 16#8E24;
   // GBK_TO_UNICODE[31474] := 16#DB6F;
   // GBK_TO_UNICODE[31475] := 16#8E25;
   // GBK_TO_UNICODE[31476] := 16#DB70;
   // GBK_TO_UNICODE[31477] := 16#8E26;
   // GBK_TO_UNICODE[31478] := 16#DB71;
   // GBK_TO_UNICODE[31479] := 16#8E27;
   // GBK_TO_UNICODE[31480] := 16#DB72;
   // GBK_TO_UNICODE[31481] := 16#8E28;
   // GBK_TO_UNICODE[31482] := 16#DB73;
   // GBK_TO_UNICODE[31483] := 16#8E2B;
   // GBK_TO_UNICODE[31484] := 16#DB74;
   // GBK_TO_UNICODE[31485] := 16#8E2D;
   // GBK_TO_UNICODE[31486] := 16#DB75;
   // GBK_TO_UNICODE[31487] := 16#8E30;
   // GBK_TO_UNICODE[31488] := 16#DB76;
   // GBK_TO_UNICODE[31489] := 16#8E32;
   // GBK_TO_UNICODE[31490] := 16#DB77;
   // GBK_TO_UNICODE[31491] := 16#8E33;
   // GBK_TO_UNICODE[31492] := 16#DB78;
   // GBK_TO_UNICODE[31493] := 16#8E34;
   // GBK_TO_UNICODE[31494] := 16#DB79;
   // GBK_TO_UNICODE[31495] := 16#8E36;
   // GBK_TO_UNICODE[31496] := 16#DB7A;
   // GBK_TO_UNICODE[31497] := 16#8E37;
   // GBK_TO_UNICODE[31498] := 16#DB7B;
   // GBK_TO_UNICODE[31499] := 16#8E38;
   // GBK_TO_UNICODE[31500] := 16#DB7C;
   // GBK_TO_UNICODE[31501] := 16#8E3B;
   // GBK_TO_UNICODE[31502] := 16#DB7D;
   // GBK_TO_UNICODE[31503] := 16#8E3C;
   // GBK_TO_UNICODE[31504] := 16#DB7E;
   // GBK_TO_UNICODE[31505] := 16#8E3E;
   // GBK_TO_UNICODE[31506] := 16#DB80;
   // GBK_TO_UNICODE[31507] := 16#8E3F;
   // GBK_TO_UNICODE[31508] := 16#DB81;
   // GBK_TO_UNICODE[31509] := 16#8E43;
   // GBK_TO_UNICODE[31510] := 16#DB82;
   // GBK_TO_UNICODE[31511] := 16#8E45;
   // GBK_TO_UNICODE[31512] := 16#DB83;
   // GBK_TO_UNICODE[31513] := 16#8E46;
   // GBK_TO_UNICODE[31514] := 16#DB84;
   // GBK_TO_UNICODE[31515] := 16#8E4C;
   // GBK_TO_UNICODE[31516] := 16#DB85;
   // GBK_TO_UNICODE[31517] := 16#8E4D;
   // GBK_TO_UNICODE[31518] := 16#DB86;
   // GBK_TO_UNICODE[31519] := 16#8E4E;
   // GBK_TO_UNICODE[31520] := 16#DB87;
   // GBK_TO_UNICODE[31521] := 16#8E4F;
   // GBK_TO_UNICODE[31522] := 16#DB88;
   // GBK_TO_UNICODE[31523] := 16#8E50;
   // GBK_TO_UNICODE[31524] := 16#DB89;
   // GBK_TO_UNICODE[31525] := 16#8E53;
   // GBK_TO_UNICODE[31526] := 16#DB8A;
   // GBK_TO_UNICODE[31527] := 16#8E54;
   // GBK_TO_UNICODE[31528] := 16#DB8B;
   // GBK_TO_UNICODE[31529] := 16#8E55;
   // GBK_TO_UNICODE[31530] := 16#DB8C;
   // GBK_TO_UNICODE[31531] := 16#8E56;
   // GBK_TO_UNICODE[31532] := 16#DB8D;
   // GBK_TO_UNICODE[31533] := 16#8E57;
   // GBK_TO_UNICODE[31534] := 16#DB8E;
   // GBK_TO_UNICODE[31535] := 16#8E58;
   // GBK_TO_UNICODE[31536] := 16#DB8F;
   // GBK_TO_UNICODE[31537] := 16#8E5A;
   // GBK_TO_UNICODE[31538] := 16#DB90;
   // GBK_TO_UNICODE[31539] := 16#8E5B;
   // GBK_TO_UNICODE[31540] := 16#DB91;
   // GBK_TO_UNICODE[31541] := 16#8E5C;
   // GBK_TO_UNICODE[31542] := 16#DB92;
   // GBK_TO_UNICODE[31543] := 16#8E5D;
   // GBK_TO_UNICODE[31544] := 16#DB93;
   // GBK_TO_UNICODE[31545] := 16#8E5E;
   // GBK_TO_UNICODE[31546] := 16#DB94;
   // GBK_TO_UNICODE[31547] := 16#8E5F;
   // GBK_TO_UNICODE[31548] := 16#DB95;
   // GBK_TO_UNICODE[31549] := 16#8E60;
   // GBK_TO_UNICODE[31550] := 16#DB96;
   // GBK_TO_UNICODE[31551] := 16#8E61;
   // GBK_TO_UNICODE[31552] := 16#DB97;
   // GBK_TO_UNICODE[31553] := 16#8E62;
   // GBK_TO_UNICODE[31554] := 16#DB98;
   // GBK_TO_UNICODE[31555] := 16#8E63;
   // GBK_TO_UNICODE[31556] := 16#DB99;
   // GBK_TO_UNICODE[31557] := 16#8E64;
   // GBK_TO_UNICODE[31558] := 16#DB9A;
   // GBK_TO_UNICODE[31559] := 16#8E65;
   // GBK_TO_UNICODE[31560] := 16#DB9B;
   // GBK_TO_UNICODE[31561] := 16#8E67;
   // GBK_TO_UNICODE[31562] := 16#DB9C;
   // GBK_TO_UNICODE[31563] := 16#8E68;
   // GBK_TO_UNICODE[31564] := 16#DB9D;
   // GBK_TO_UNICODE[31565] := 16#8E6A;
   // GBK_TO_UNICODE[31566] := 16#DB9E;
   // GBK_TO_UNICODE[31567] := 16#8E6B;
   // GBK_TO_UNICODE[31568] := 16#DB9F;
   // GBK_TO_UNICODE[31569] := 16#8E6E;
   // GBK_TO_UNICODE[31570] := 16#DBA0;
   // GBK_TO_UNICODE[31571] := 16#8E71;
   // GBK_TO_UNICODE[31572] := 16#DBA1;
   // GBK_TO_UNICODE[31573] := 16#90B8;
   // GBK_TO_UNICODE[31574] := 16#DBA2;
   // GBK_TO_UNICODE[31575] := 16#90B0;
   // GBK_TO_UNICODE[31576] := 16#DBA3;
   // GBK_TO_UNICODE[31577] := 16#90CF;
   // GBK_TO_UNICODE[31578] := 16#DBA4;
   // GBK_TO_UNICODE[31579] := 16#90C5;
   // GBK_TO_UNICODE[31580] := 16#DBA5;
   // GBK_TO_UNICODE[31581] := 16#90BE;
   // GBK_TO_UNICODE[31582] := 16#DBA6;
   // GBK_TO_UNICODE[31583] := 16#90D0;
   // GBK_TO_UNICODE[31584] := 16#DBA7;
   // GBK_TO_UNICODE[31585] := 16#90C4;
   // GBK_TO_UNICODE[31586] := 16#DBA8;
   // GBK_TO_UNICODE[31587] := 16#90C7;
   // GBK_TO_UNICODE[31588] := 16#DBA9;
   // GBK_TO_UNICODE[31589] := 16#90D3;
   // GBK_TO_UNICODE[31590] := 16#DBAA;
   // GBK_TO_UNICODE[31591] := 16#90E6;
   // GBK_TO_UNICODE[31592] := 16#DBAB;
   // GBK_TO_UNICODE[31593] := 16#90E2;
   // GBK_TO_UNICODE[31594] := 16#DBAC;
   // GBK_TO_UNICODE[31595] := 16#90DC;
   // GBK_TO_UNICODE[31596] := 16#DBAD;
   // GBK_TO_UNICODE[31597] := 16#90D7;
   // GBK_TO_UNICODE[31598] := 16#DBAE;
   // GBK_TO_UNICODE[31599] := 16#90DB;
   // GBK_TO_UNICODE[31600] := 16#DBAF;
   // GBK_TO_UNICODE[31601] := 16#90EB;
   // GBK_TO_UNICODE[31602] := 16#DBB0;
   // GBK_TO_UNICODE[31603] := 16#90EF;
   // GBK_TO_UNICODE[31604] := 16#DBB1;
   // GBK_TO_UNICODE[31605] := 16#90FE;
   // GBK_TO_UNICODE[31606] := 16#DBB2;
   // GBK_TO_UNICODE[31607] := 16#9104;
   // GBK_TO_UNICODE[31608] := 16#DBB3;
   // GBK_TO_UNICODE[31609] := 16#9122;
   // GBK_TO_UNICODE[31610] := 16#DBB4;
   // GBK_TO_UNICODE[31611] := 16#911E;
   // GBK_TO_UNICODE[31612] := 16#DBB5;
   // GBK_TO_UNICODE[31613] := 16#9123;
   // GBK_TO_UNICODE[31614] := 16#DBB6;
   // GBK_TO_UNICODE[31615] := 16#9131;
   // GBK_TO_UNICODE[31616] := 16#DBB7;
   // GBK_TO_UNICODE[31617] := 16#912F;
   // GBK_TO_UNICODE[31618] := 16#DBB8;
   // GBK_TO_UNICODE[31619] := 16#9139;
   // GBK_TO_UNICODE[31620] := 16#DBB9;
   // GBK_TO_UNICODE[31621] := 16#9143;
   // GBK_TO_UNICODE[31622] := 16#DBBA;
   // GBK_TO_UNICODE[31623] := 16#9146;
   // GBK_TO_UNICODE[31624] := 16#DBBB;
   // GBK_TO_UNICODE[31625] := 16#520D;
   // GBK_TO_UNICODE[31626] := 16#DBBC;
   // GBK_TO_UNICODE[31627] := 16#5942;
   // GBK_TO_UNICODE[31628] := 16#DBBD;
   // GBK_TO_UNICODE[31629] := 16#52A2;
   // GBK_TO_UNICODE[31630] := 16#DBBE;
   // GBK_TO_UNICODE[31631] := 16#52AC;
   // GBK_TO_UNICODE[31632] := 16#DBBF;
   // GBK_TO_UNICODE[31633] := 16#52AD;
   // GBK_TO_UNICODE[31634] := 16#DBC0;
   // GBK_TO_UNICODE[31635] := 16#52BE;
   // GBK_TO_UNICODE[31636] := 16#DBC1;
   // GBK_TO_UNICODE[31637] := 16#54FF;
   // GBK_TO_UNICODE[31638] := 16#DBC2;
   // GBK_TO_UNICODE[31639] := 16#52D0;
   // GBK_TO_UNICODE[31640] := 16#DBC3;
   // GBK_TO_UNICODE[31641] := 16#52D6;
   // GBK_TO_UNICODE[31642] := 16#DBC4;
   // GBK_TO_UNICODE[31643] := 16#52F0;
   // GBK_TO_UNICODE[31644] := 16#DBC5;
   // GBK_TO_UNICODE[31645] := 16#53DF;
   // GBK_TO_UNICODE[31646] := 16#DBC6;
   // GBK_TO_UNICODE[31647] := 16#71EE;
   // GBK_TO_UNICODE[31648] := 16#DBC7;
   // GBK_TO_UNICODE[31649] := 16#77CD;
   // GBK_TO_UNICODE[31650] := 16#DBC8;
   // GBK_TO_UNICODE[31651] := 16#5EF4;
   // GBK_TO_UNICODE[31652] := 16#DBC9;
   // GBK_TO_UNICODE[31653] := 16#51F5;
   // GBK_TO_UNICODE[31654] := 16#DBCA;
   // GBK_TO_UNICODE[31655] := 16#51FC;
   // GBK_TO_UNICODE[31656] := 16#DBCB;
   // GBK_TO_UNICODE[31657] := 16#9B2F;
   // GBK_TO_UNICODE[31658] := 16#DBCC;
   // GBK_TO_UNICODE[31659] := 16#53B6;
   // GBK_TO_UNICODE[31660] := 16#DBCD;
   // GBK_TO_UNICODE[31661] := 16#5F01;
   // GBK_TO_UNICODE[31662] := 16#DBCE;
   // GBK_TO_UNICODE[31663] := 16#755A;
   // GBK_TO_UNICODE[31664] := 16#DBCF;
   // GBK_TO_UNICODE[31665] := 16#5DEF;
   // GBK_TO_UNICODE[31666] := 16#DBD0;
   // GBK_TO_UNICODE[31667] := 16#574C;
   // GBK_TO_UNICODE[31668] := 16#DBD1;
   // GBK_TO_UNICODE[31669] := 16#57A9;
   // GBK_TO_UNICODE[31670] := 16#DBD2;
   // GBK_TO_UNICODE[31671] := 16#57A1;
   // GBK_TO_UNICODE[31672] := 16#DBD3;
   // GBK_TO_UNICODE[31673] := 16#587E;
   // GBK_TO_UNICODE[31674] := 16#DBD4;
   // GBK_TO_UNICODE[31675] := 16#58BC;
   // GBK_TO_UNICODE[31676] := 16#DBD5;
   // GBK_TO_UNICODE[31677] := 16#58C5;
   // GBK_TO_UNICODE[31678] := 16#DBD6;
   // GBK_TO_UNICODE[31679] := 16#58D1;
   // GBK_TO_UNICODE[31680] := 16#DBD7;
   // GBK_TO_UNICODE[31681] := 16#5729;
   // GBK_TO_UNICODE[31682] := 16#DBD8;
   // GBK_TO_UNICODE[31683] := 16#572C;
   // GBK_TO_UNICODE[31684] := 16#DBD9;
   // GBK_TO_UNICODE[31685] := 16#572A;
   // GBK_TO_UNICODE[31686] := 16#DBDA;
   // GBK_TO_UNICODE[31687] := 16#5733;
   // GBK_TO_UNICODE[31688] := 16#DBDB;
   // GBK_TO_UNICODE[31689] := 16#5739;
   // GBK_TO_UNICODE[31690] := 16#DBDC;
   // GBK_TO_UNICODE[31691] := 16#572E;
   // GBK_TO_UNICODE[31692] := 16#DBDD;
   // GBK_TO_UNICODE[31693] := 16#572F;
   // GBK_TO_UNICODE[31694] := 16#DBDE;
   // GBK_TO_UNICODE[31695] := 16#575C;
   // GBK_TO_UNICODE[31696] := 16#DBDF;
   // GBK_TO_UNICODE[31697] := 16#573B;
   // GBK_TO_UNICODE[31698] := 16#DBE0;
   // GBK_TO_UNICODE[31699] := 16#5742;
   // GBK_TO_UNICODE[31700] := 16#DBE1;
   // GBK_TO_UNICODE[31701] := 16#5769;
   // GBK_TO_UNICODE[31702] := 16#DBE2;
   // GBK_TO_UNICODE[31703] := 16#5785;
   // GBK_TO_UNICODE[31704] := 16#DBE3;
   // GBK_TO_UNICODE[31705] := 16#576B;
   // GBK_TO_UNICODE[31706] := 16#DBE4;
   // GBK_TO_UNICODE[31707] := 16#5786;
   // GBK_TO_UNICODE[31708] := 16#DBE5;
   // GBK_TO_UNICODE[31709] := 16#577C;
   // GBK_TO_UNICODE[31710] := 16#DBE6;
   // GBK_TO_UNICODE[31711] := 16#577B;
   // GBK_TO_UNICODE[31712] := 16#DBE7;
   // GBK_TO_UNICODE[31713] := 16#5768;
   // GBK_TO_UNICODE[31714] := 16#DBE8;
   // GBK_TO_UNICODE[31715] := 16#576D;
   // GBK_TO_UNICODE[31716] := 16#DBE9;
   // GBK_TO_UNICODE[31717] := 16#5776;
   // GBK_TO_UNICODE[31718] := 16#DBEA;
   // GBK_TO_UNICODE[31719] := 16#5773;
   // GBK_TO_UNICODE[31720] := 16#DBEB;
   // GBK_TO_UNICODE[31721] := 16#57AD;
   // GBK_TO_UNICODE[31722] := 16#DBEC;
   // GBK_TO_UNICODE[31723] := 16#57A4;
   // GBK_TO_UNICODE[31724] := 16#DBED;
   // GBK_TO_UNICODE[31725] := 16#578C;
   // GBK_TO_UNICODE[31726] := 16#DBEE;
   // GBK_TO_UNICODE[31727] := 16#57B2;
   // GBK_TO_UNICODE[31728] := 16#DBEF;
   // GBK_TO_UNICODE[31729] := 16#57CF;
   // GBK_TO_UNICODE[31730] := 16#DBF0;
   // GBK_TO_UNICODE[31731] := 16#57A7;
   // GBK_TO_UNICODE[31732] := 16#DBF1;
   // GBK_TO_UNICODE[31733] := 16#57B4;
   // GBK_TO_UNICODE[31734] := 16#DBF2;
   // GBK_TO_UNICODE[31735] := 16#5793;
   // GBK_TO_UNICODE[31736] := 16#DBF3;
   // GBK_TO_UNICODE[31737] := 16#57A0;
   // GBK_TO_UNICODE[31738] := 16#DBF4;
   // GBK_TO_UNICODE[31739] := 16#57D5;
   // GBK_TO_UNICODE[31740] := 16#DBF5;
   // GBK_TO_UNICODE[31741] := 16#57D8;
   // GBK_TO_UNICODE[31742] := 16#DBF6;
   // GBK_TO_UNICODE[31743] := 16#57DA;
   // GBK_TO_UNICODE[31744] := 16#DBF7;
   // GBK_TO_UNICODE[31745] := 16#57D9;
   // GBK_TO_UNICODE[31746] := 16#DBF8;
   // GBK_TO_UNICODE[31747] := 16#57D2;
   // GBK_TO_UNICODE[31748] := 16#DBF9;
   // GBK_TO_UNICODE[31749] := 16#57B8;
   // GBK_TO_UNICODE[31750] := 16#DBFA;
   // GBK_TO_UNICODE[31751] := 16#57F4;
   // GBK_TO_UNICODE[31752] := 16#DBFB;
   // GBK_TO_UNICODE[31753] := 16#57EF;
   // GBK_TO_UNICODE[31754] := 16#DBFC;
   // GBK_TO_UNICODE[31755] := 16#57F8;
   // GBK_TO_UNICODE[31756] := 16#DBFD;
   // GBK_TO_UNICODE[31757] := 16#57E4;
   // GBK_TO_UNICODE[31758] := 16#DBFE;
   // GBK_TO_UNICODE[31759] := 16#57DD;
   // GBK_TO_UNICODE[31760] := 16#DC40;
   // GBK_TO_UNICODE[31761] := 16#8E73;
   // GBK_TO_UNICODE[31762] := 16#DC41;
   // GBK_TO_UNICODE[31763] := 16#8E75;
   // GBK_TO_UNICODE[31764] := 16#DC42;
   // GBK_TO_UNICODE[31765] := 16#8E77;
   // GBK_TO_UNICODE[31766] := 16#DC43;
   // GBK_TO_UNICODE[31767] := 16#8E78;
   // GBK_TO_UNICODE[31768] := 16#DC44;
   // GBK_TO_UNICODE[31769] := 16#8E79;
   // GBK_TO_UNICODE[31770] := 16#DC45;
   // GBK_TO_UNICODE[31771] := 16#8E7A;
   // GBK_TO_UNICODE[31772] := 16#DC46;
   // GBK_TO_UNICODE[31773] := 16#8E7B;
   // GBK_TO_UNICODE[31774] := 16#DC47;
   // GBK_TO_UNICODE[31775] := 16#8E7D;
   // GBK_TO_UNICODE[31776] := 16#DC48;
   // GBK_TO_UNICODE[31777] := 16#8E7E;
   // GBK_TO_UNICODE[31778] := 16#DC49;
   // GBK_TO_UNICODE[31779] := 16#8E80;
   // GBK_TO_UNICODE[31780] := 16#DC4A;
   // GBK_TO_UNICODE[31781] := 16#8E82;
   // GBK_TO_UNICODE[31782] := 16#DC4B;
   // GBK_TO_UNICODE[31783] := 16#8E83;
   // GBK_TO_UNICODE[31784] := 16#DC4C;
   // GBK_TO_UNICODE[31785] := 16#8E84;
   // GBK_TO_UNICODE[31786] := 16#DC4D;
   // GBK_TO_UNICODE[31787] := 16#8E86;
   // GBK_TO_UNICODE[31788] := 16#DC4E;
   // GBK_TO_UNICODE[31789] := 16#8E88;
   // GBK_TO_UNICODE[31790] := 16#DC4F;
   // GBK_TO_UNICODE[31791] := 16#8E89;
   // GBK_TO_UNICODE[31792] := 16#DC50;
   // GBK_TO_UNICODE[31793] := 16#8E8A;
   // GBK_TO_UNICODE[31794] := 16#DC51;
   // GBK_TO_UNICODE[31795] := 16#8E8B;
   // GBK_TO_UNICODE[31796] := 16#DC52;
   // GBK_TO_UNICODE[31797] := 16#8E8C;
   // GBK_TO_UNICODE[31798] := 16#DC53;
   // GBK_TO_UNICODE[31799] := 16#8E8D;
   // GBK_TO_UNICODE[31800] := 16#DC54;
   // GBK_TO_UNICODE[31801] := 16#8E8E;
   // GBK_TO_UNICODE[31802] := 16#DC55;
   // GBK_TO_UNICODE[31803] := 16#8E91;
   // GBK_TO_UNICODE[31804] := 16#DC56;
   // GBK_TO_UNICODE[31805] := 16#8E92;
   // GBK_TO_UNICODE[31806] := 16#DC57;
   // GBK_TO_UNICODE[31807] := 16#8E93;
   // GBK_TO_UNICODE[31808] := 16#DC58;
   // GBK_TO_UNICODE[31809] := 16#8E95;
   // GBK_TO_UNICODE[31810] := 16#DC59;
   // GBK_TO_UNICODE[31811] := 16#8E96;
   // GBK_TO_UNICODE[31812] := 16#DC5A;
   // GBK_TO_UNICODE[31813] := 16#8E97;
   // GBK_TO_UNICODE[31814] := 16#DC5B;
   // GBK_TO_UNICODE[31815] := 16#8E98;
   // GBK_TO_UNICODE[31816] := 16#DC5C;
   // GBK_TO_UNICODE[31817] := 16#8E99;
   // GBK_TO_UNICODE[31818] := 16#DC5D;
   // GBK_TO_UNICODE[31819] := 16#8E9A;
   // GBK_TO_UNICODE[31820] := 16#DC5E;
   // GBK_TO_UNICODE[31821] := 16#8E9B;
   // GBK_TO_UNICODE[31822] := 16#DC5F;
   // GBK_TO_UNICODE[31823] := 16#8E9D;
   // GBK_TO_UNICODE[31824] := 16#DC60;
   // GBK_TO_UNICODE[31825] := 16#8E9F;
   // GBK_TO_UNICODE[31826] := 16#DC61;
   // GBK_TO_UNICODE[31827] := 16#8EA0;
   // GBK_TO_UNICODE[31828] := 16#DC62;
   // GBK_TO_UNICODE[31829] := 16#8EA1;
   // GBK_TO_UNICODE[31830] := 16#DC63;
   // GBK_TO_UNICODE[31831] := 16#8EA2;
   // GBK_TO_UNICODE[31832] := 16#DC64;
   // GBK_TO_UNICODE[31833] := 16#8EA3;
   // GBK_TO_UNICODE[31834] := 16#DC65;
   // GBK_TO_UNICODE[31835] := 16#8EA4;
   // GBK_TO_UNICODE[31836] := 16#DC66;
   // GBK_TO_UNICODE[31837] := 16#8EA5;
   // GBK_TO_UNICODE[31838] := 16#DC67;
   // GBK_TO_UNICODE[31839] := 16#8EA6;
   // GBK_TO_UNICODE[31840] := 16#DC68;
   // GBK_TO_UNICODE[31841] := 16#8EA7;
   // GBK_TO_UNICODE[31842] := 16#DC69;
   // GBK_TO_UNICODE[31843] := 16#8EA8;
   // GBK_TO_UNICODE[31844] := 16#DC6A;
   // GBK_TO_UNICODE[31845] := 16#8EA9;
   // GBK_TO_UNICODE[31846] := 16#DC6B;
   // GBK_TO_UNICODE[31847] := 16#8EAA;
   // GBK_TO_UNICODE[31848] := 16#DC6C;
   // GBK_TO_UNICODE[31849] := 16#8EAD;
   // GBK_TO_UNICODE[31850] := 16#DC6D;
   // GBK_TO_UNICODE[31851] := 16#8EAE;
   // GBK_TO_UNICODE[31852] := 16#DC6E;
   // GBK_TO_UNICODE[31853] := 16#8EB0;
   // GBK_TO_UNICODE[31854] := 16#DC6F;
   // GBK_TO_UNICODE[31855] := 16#8EB1;
   // GBK_TO_UNICODE[31856] := 16#DC70;
   // GBK_TO_UNICODE[31857] := 16#8EB3;
   // GBK_TO_UNICODE[31858] := 16#DC71;
   // GBK_TO_UNICODE[31859] := 16#8EB4;
   // GBK_TO_UNICODE[31860] := 16#DC72;
   // GBK_TO_UNICODE[31861] := 16#8EB5;
   // GBK_TO_UNICODE[31862] := 16#DC73;
   // GBK_TO_UNICODE[31863] := 16#8EB6;
   // GBK_TO_UNICODE[31864] := 16#DC74;
   // GBK_TO_UNICODE[31865] := 16#8EB7;
   // GBK_TO_UNICODE[31866] := 16#DC75;
   // GBK_TO_UNICODE[31867] := 16#8EB8;
   // GBK_TO_UNICODE[31868] := 16#DC76;
   // GBK_TO_UNICODE[31869] := 16#8EB9;
   // GBK_TO_UNICODE[31870] := 16#DC77;
   // GBK_TO_UNICODE[31871] := 16#8EBB;
   // GBK_TO_UNICODE[31872] := 16#DC78;
   // GBK_TO_UNICODE[31873] := 16#8EBC;
   // GBK_TO_UNICODE[31874] := 16#DC79;
   // GBK_TO_UNICODE[31875] := 16#8EBD;
   // GBK_TO_UNICODE[31876] := 16#DC7A;
   // GBK_TO_UNICODE[31877] := 16#8EBE;
   // GBK_TO_UNICODE[31878] := 16#DC7B;
   // GBK_TO_UNICODE[31879] := 16#8EBF;
   // GBK_TO_UNICODE[31880] := 16#DC7C;
   // GBK_TO_UNICODE[31881] := 16#8EC0;
   // GBK_TO_UNICODE[31882] := 16#DC7D;
   // GBK_TO_UNICODE[31883] := 16#8EC1;
   // GBK_TO_UNICODE[31884] := 16#DC7E;
   // GBK_TO_UNICODE[31885] := 16#8EC2;
   // GBK_TO_UNICODE[31886] := 16#DC80;
   // GBK_TO_UNICODE[31887] := 16#8EC3;
   // GBK_TO_UNICODE[31888] := 16#DC81;
   // GBK_TO_UNICODE[31889] := 16#8EC4;
   // GBK_TO_UNICODE[31890] := 16#DC82;
   // GBK_TO_UNICODE[31891] := 16#8EC5;
   // GBK_TO_UNICODE[31892] := 16#DC83;
   // GBK_TO_UNICODE[31893] := 16#8EC6;
   // GBK_TO_UNICODE[31894] := 16#DC84;
   // GBK_TO_UNICODE[31895] := 16#8EC7;
   // GBK_TO_UNICODE[31896] := 16#DC85;
   // GBK_TO_UNICODE[31897] := 16#8EC8;
   // GBK_TO_UNICODE[31898] := 16#DC86;
   // GBK_TO_UNICODE[31899] := 16#8EC9;
   // GBK_TO_UNICODE[31900] := 16#DC87;
   // GBK_TO_UNICODE[31901] := 16#8ECA;
   // GBK_TO_UNICODE[31902] := 16#DC88;
   // GBK_TO_UNICODE[31903] := 16#8ECB;
   // GBK_TO_UNICODE[31904] := 16#DC89;
   // GBK_TO_UNICODE[31905] := 16#8ECC;
   // GBK_TO_UNICODE[31906] := 16#DC8A;
   // GBK_TO_UNICODE[31907] := 16#8ECD;
   // GBK_TO_UNICODE[31908] := 16#DC8B;
   // GBK_TO_UNICODE[31909] := 16#8ECF;
   // GBK_TO_UNICODE[31910] := 16#DC8C;
   // GBK_TO_UNICODE[31911] := 16#8ED0;
   // GBK_TO_UNICODE[31912] := 16#DC8D;
   // GBK_TO_UNICODE[31913] := 16#8ED1;
   // GBK_TO_UNICODE[31914] := 16#DC8E;
   // GBK_TO_UNICODE[31915] := 16#8ED2;
   // GBK_TO_UNICODE[31916] := 16#DC8F;
   // GBK_TO_UNICODE[31917] := 16#8ED3;
   // GBK_TO_UNICODE[31918] := 16#DC90;
   // GBK_TO_UNICODE[31919] := 16#8ED4;
   // GBK_TO_UNICODE[31920] := 16#DC91;
   // GBK_TO_UNICODE[31921] := 16#8ED5;
   // GBK_TO_UNICODE[31922] := 16#DC92;
   // GBK_TO_UNICODE[31923] := 16#8ED6;
   // GBK_TO_UNICODE[31924] := 16#DC93;
   // GBK_TO_UNICODE[31925] := 16#8ED7;
   // GBK_TO_UNICODE[31926] := 16#DC94;
   // GBK_TO_UNICODE[31927] := 16#8ED8;
   // GBK_TO_UNICODE[31928] := 16#DC95;
   // GBK_TO_UNICODE[31929] := 16#8ED9;
   // GBK_TO_UNICODE[31930] := 16#DC96;
   // GBK_TO_UNICODE[31931] := 16#8EDA;
   // GBK_TO_UNICODE[31932] := 16#DC97;
   // GBK_TO_UNICODE[31933] := 16#8EDB;
   // GBK_TO_UNICODE[31934] := 16#DC98;
   // GBK_TO_UNICODE[31935] := 16#8EDC;
   // GBK_TO_UNICODE[31936] := 16#DC99;
   // GBK_TO_UNICODE[31937] := 16#8EDD;
   // GBK_TO_UNICODE[31938] := 16#DC9A;
   // GBK_TO_UNICODE[31939] := 16#8EDE;
   // GBK_TO_UNICODE[31940] := 16#DC9B;
   // GBK_TO_UNICODE[31941] := 16#8EDF;
   // GBK_TO_UNICODE[31942] := 16#DC9C;
   // GBK_TO_UNICODE[31943] := 16#8EE0;
   // GBK_TO_UNICODE[31944] := 16#DC9D;
   // GBK_TO_UNICODE[31945] := 16#8EE1;
   // GBK_TO_UNICODE[31946] := 16#DC9E;
   // GBK_TO_UNICODE[31947] := 16#8EE2;
   // GBK_TO_UNICODE[31948] := 16#DC9F;
   // GBK_TO_UNICODE[31949] := 16#8EE3;
   // GBK_TO_UNICODE[31950] := 16#DCA0;
   // GBK_TO_UNICODE[31951] := 16#8EE4;
   // GBK_TO_UNICODE[31952] := 16#DCA1;
   // GBK_TO_UNICODE[31953] := 16#580B;
   // GBK_TO_UNICODE[31954] := 16#DCA2;
   // GBK_TO_UNICODE[31955] := 16#580D;
   // GBK_TO_UNICODE[31956] := 16#DCA3;
   // GBK_TO_UNICODE[31957] := 16#57FD;
   // GBK_TO_UNICODE[31958] := 16#DCA4;
   // GBK_TO_UNICODE[31959] := 16#57ED;
   // GBK_TO_UNICODE[31960] := 16#DCA5;
   // GBK_TO_UNICODE[31961] := 16#5800;
   // GBK_TO_UNICODE[31962] := 16#DCA6;
   // GBK_TO_UNICODE[31963] := 16#581E;
   // GBK_TO_UNICODE[31964] := 16#DCA7;
   // GBK_TO_UNICODE[31965] := 16#5819;
   // GBK_TO_UNICODE[31966] := 16#DCA8;
   // GBK_TO_UNICODE[31967] := 16#5844;
   // GBK_TO_UNICODE[31968] := 16#DCA9;
   // GBK_TO_UNICODE[31969] := 16#5820;
   // GBK_TO_UNICODE[31970] := 16#DCAA;
   // GBK_TO_UNICODE[31971] := 16#5865;
   // GBK_TO_UNICODE[31972] := 16#DCAB;
   // GBK_TO_UNICODE[31973] := 16#586C;
   // GBK_TO_UNICODE[31974] := 16#DCAC;
   // GBK_TO_UNICODE[31975] := 16#5881;
   // GBK_TO_UNICODE[31976] := 16#DCAD;
   // GBK_TO_UNICODE[31977] := 16#5889;
   // GBK_TO_UNICODE[31978] := 16#DCAE;
   // GBK_TO_UNICODE[31979] := 16#589A;
   // GBK_TO_UNICODE[31980] := 16#DCAF;
   // GBK_TO_UNICODE[31981] := 16#5880;
   // GBK_TO_UNICODE[31982] := 16#DCB0;
   // GBK_TO_UNICODE[31983] := 16#99A8;
   // GBK_TO_UNICODE[31984] := 16#DCB1;
   // GBK_TO_UNICODE[31985] := 16#9F19;
   // GBK_TO_UNICODE[31986] := 16#DCB2;
   // GBK_TO_UNICODE[31987] := 16#61FF;
   // GBK_TO_UNICODE[31988] := 16#DCB3;
   // GBK_TO_UNICODE[31989] := 16#8279;
   // GBK_TO_UNICODE[31990] := 16#DCB4;
   // GBK_TO_UNICODE[31991] := 16#827D;
   // GBK_TO_UNICODE[31992] := 16#DCB5;
   // GBK_TO_UNICODE[31993] := 16#827F;
   // GBK_TO_UNICODE[31994] := 16#DCB6;
   // GBK_TO_UNICODE[31995] := 16#828F;
   // GBK_TO_UNICODE[31996] := 16#DCB7;
   // GBK_TO_UNICODE[31997] := 16#828A;
   // GBK_TO_UNICODE[31998] := 16#DCB8;
   // GBK_TO_UNICODE[31999] := 16#82A8;
   // GBK_TO_UNICODE[32000] := 16#DCB9;
   // GBK_TO_UNICODE[32001] := 16#8284;
   // GBK_TO_UNICODE[32002] := 16#DCBA;
   // GBK_TO_UNICODE[32003] := 16#828E;
   // GBK_TO_UNICODE[32004] := 16#DCBB;
   // GBK_TO_UNICODE[32005] := 16#8291;
   // GBK_TO_UNICODE[32006] := 16#DCBC;
   // GBK_TO_UNICODE[32007] := 16#8297;
   // GBK_TO_UNICODE[32008] := 16#DCBD;
   // GBK_TO_UNICODE[32009] := 16#8299;
   // GBK_TO_UNICODE[32010] := 16#DCBE;
   // GBK_TO_UNICODE[32011] := 16#82AB;
   // GBK_TO_UNICODE[32012] := 16#DCBF;
   // GBK_TO_UNICODE[32013] := 16#82B8;
   // GBK_TO_UNICODE[32014] := 16#DCC0;
   // GBK_TO_UNICODE[32015] := 16#82BE;
   // GBK_TO_UNICODE[32016] := 16#DCC1;
   // GBK_TO_UNICODE[32017] := 16#82B0;
   // GBK_TO_UNICODE[32018] := 16#DCC2;
   // GBK_TO_UNICODE[32019] := 16#82C8;
   // GBK_TO_UNICODE[32020] := 16#DCC3;
   // GBK_TO_UNICODE[32021] := 16#82CA;
   // GBK_TO_UNICODE[32022] := 16#DCC4;
   // GBK_TO_UNICODE[32023] := 16#82E3;
   // GBK_TO_UNICODE[32024] := 16#DCC5;
   // GBK_TO_UNICODE[32025] := 16#8298;
   // GBK_TO_UNICODE[32026] := 16#DCC6;
   // GBK_TO_UNICODE[32027] := 16#82B7;
   // GBK_TO_UNICODE[32028] := 16#DCC7;
   // GBK_TO_UNICODE[32029] := 16#82AE;
   // GBK_TO_UNICODE[32030] := 16#DCC8;
   // GBK_TO_UNICODE[32031] := 16#82CB;
   // GBK_TO_UNICODE[32032] := 16#DCC9;
   // GBK_TO_UNICODE[32033] := 16#82CC;
   // GBK_TO_UNICODE[32034] := 16#DCCA;
   // GBK_TO_UNICODE[32035] := 16#82C1;
   // GBK_TO_UNICODE[32036] := 16#DCCB;
   // GBK_TO_UNICODE[32037] := 16#82A9;
   // GBK_TO_UNICODE[32038] := 16#DCCC;
   // GBK_TO_UNICODE[32039] := 16#82B4;
   // GBK_TO_UNICODE[32040] := 16#DCCD;
   // GBK_TO_UNICODE[32041] := 16#82A1;
   // GBK_TO_UNICODE[32042] := 16#DCCE;
   // GBK_TO_UNICODE[32043] := 16#82AA;
   // GBK_TO_UNICODE[32044] := 16#DCCF;
   // GBK_TO_UNICODE[32045] := 16#829F;
   // GBK_TO_UNICODE[32046] := 16#DCD0;
   // GBK_TO_UNICODE[32047] := 16#82C4;
   // GBK_TO_UNICODE[32048] := 16#DCD1;
   // GBK_TO_UNICODE[32049] := 16#82CE;
   // GBK_TO_UNICODE[32050] := 16#DCD2;
   // GBK_TO_UNICODE[32051] := 16#82A4;
   // GBK_TO_UNICODE[32052] := 16#DCD3;
   // GBK_TO_UNICODE[32053] := 16#82E1;
   // GBK_TO_UNICODE[32054] := 16#DCD4;
   // GBK_TO_UNICODE[32055] := 16#8309;
   // GBK_TO_UNICODE[32056] := 16#DCD5;
   // GBK_TO_UNICODE[32057] := 16#82F7;
   // GBK_TO_UNICODE[32058] := 16#DCD6;
   // GBK_TO_UNICODE[32059] := 16#82E4;
   // GBK_TO_UNICODE[32060] := 16#DCD7;
   // GBK_TO_UNICODE[32061] := 16#830F;
   // GBK_TO_UNICODE[32062] := 16#DCD8;
   // GBK_TO_UNICODE[32063] := 16#8307;
   // GBK_TO_UNICODE[32064] := 16#DCD9;
   // GBK_TO_UNICODE[32065] := 16#82DC;
   // GBK_TO_UNICODE[32066] := 16#DCDA;
   // GBK_TO_UNICODE[32067] := 16#82F4;
